FUNCTION_BLOCK "HF3_FJPG_FB2771"	// FB 2771
VERSION : 0.1
VAR
  PT : TIME  := T#45S;
  AP22_WP14 : FB 2772;
END_VAR
BEGIN
NETWORK
TITLE = AP22-wp14
      A     "EPS11_QJSS_UEF_Opd";
      =     L 0.0;
      BLD   103;
      A     "EPS11_QJSS_UEB_Opd";
      =     L 0.1;
      BLD   103;
      A     "EPS11_QJSS_DHF_Opd";
      =     L 0.2;
      BLD   103;
      A     DB7004.DBX 2630.0;
      =     L 0.4;
      BLD   103;
      A     DB7004.DBX 2630.1;
      =     L 0.5;
      BLD   103;
      BLD   14;
      =     L 7.0;
      L     DINO;
      T     LW 5;
      CDB;
      OPN   DI [LW 5];
      TAR2  LD 1;
      OPN   DI 6001;
      L     DIW 170;
      OPN   DI [LW 5];
      T     #AP22_WP14.SCtrl;
      OPN   DI 7004;
      L     DIW 840;
      OPN   DI [LW 5];
      T     #AP22_WP14.H_P_ALL_Ctrl;
      A     L 0.0;
      =     #AP22_WP14.DI_LR;
      A     L 0.1;
      =     #AP22_WP14.DI_Run;
      A     L 0.2;
      =     #AP22_WP14.DI_Stp;
      A     L 0.4;
      =     #AP22_WP14.FireAlarm;
      A     L 0.5;
      =     #AP22_WP14.BlockAlarm;
      BLD   11;
      L     W#16#1002;
      T     LW 10;
      L     2;
      T     LW 12;
      L     7004;
      T     LW 14;
      L     P#DBX 592.0;
      T     LD 16;
      L     W#16#1002;
      T     LW 20;
      L     2;
      T     LW 22;
      L     DINO;
      T     LW 24;
      +AR2  P#12.0;
      TAR2;
      LAR2  LD 1;
      T     LD 26;
      UC    "BLKMOV";
      {     P#L 10.0, P#L 8.0, P#L 20.0 };
      BLD   11;
      L     W#16#1002;
      T     LW 10;
      L     2;
      T     LW 12;
      L     7004;
      T     LW 14;
      L     P#DBX 966.0;
      T     LD 16;
      L     W#16#1002;
      T     LW 20;
      L     2;
      T     LW 22;
      L     DINO;
      T     LW 24;
      +AR2  P#14.0;
      TAR2;
      LAR2  LD 1;
      T     LD 26;
      UC    "BLKMOV";
      {     P#L 10.0, P#L 8.0, P#L 20.0 };
      L     DBD [AR2,P#0.0];
      T     #AP22_WP14.PT1;
      +AR2  P#4.0;
      UC    "HF3_FJPG_FB2772";
      LAR2  LD 1;
      A     #AP22_WP14.DO_Run;
      =     Q 2.0;
      A     #AP22_WP14.DO_Stp;
      =     Q 2.1;
      L     #AP22_WP14.ToHMI;
      OPN   DI 6002;
      T     DIW 1110;
      OPN   DI [LW 5];
      CDB;
      BLD   15;
      NOP   0;
NETWORK
TITLE = AP_B02
END_FUNCTION_BLOCK

FUNCTION_BLOCK "HF3_FJPG_FB2772"	// FB 2772
VERSION : 0.1
VAR_INPUT
  SCtrl : WORD ;	//0.单控1.模控2.单控启动3.单控停止5.超时复位11.运行次数清零12.故障清零13.
  H_P_ALL_Ctrl : WORD ;	//全局命令
  DI_LR : BOOL ;	//远程/就地
  DI_Run : BOOL ;	//风机盘管运行反馈
  DI_Stp : BOOL ;	//风机盘管停止反馈
  Stop : BOOL ;	//连锁信号
  FireAlarm : BOOL ;	//火灾信号
  BlockAlarm : BOOL ;	//阻塞信号
  MCtrl : ARRAY  [0 .. 3 ] OF //模式控制
  BOOL ;
  Mode : ARRAY  [0 .. 15 ] OF //模式执行状态
  BOOL ;
  ALL : ARRAY  [0 .. 15 ] OF //单系统命令
  BOOL ;
  PT1 : TIME ;	//设备动作超时
END_VAR
VAR_OUTPUT
  DO_Run : BOOL ;	//开阀控制
  DO_Stp : BOOL ;	//关阀控制
  ToHMI : WORD ;	//给上位信号
END_VAR
VAR
  SCtrl_Temp : ARRAY  [0 .. 15 ] OF //1.模控2.单控启动3.单控停止5.超时复位11.运行次数清零12.故障清零13.
  BOOL ;
  DI_Temp : ARRAY  [0 .. 15 ] OF BOOL ;
  DO_Temp : ARRAY  [0 .. 15 ] OF BOOL ;
  H_P_ALL_Ctrl_Temp : ARRAY  [0 .. 15 ] OF BOOL ;
  Ctrl : ARRAY  [0 .. 15 ] OF BOOL ;
  TON1 : SFB 4;
  SFlag : BOOL ;
  QTout : BOOL ;
  Timeout : BOOL ;	//设备动作超时
  Refuse : BOOL ;	//模式不符
  McFlag : BOOL ;	//检修牌
END_VAR
BEGIN
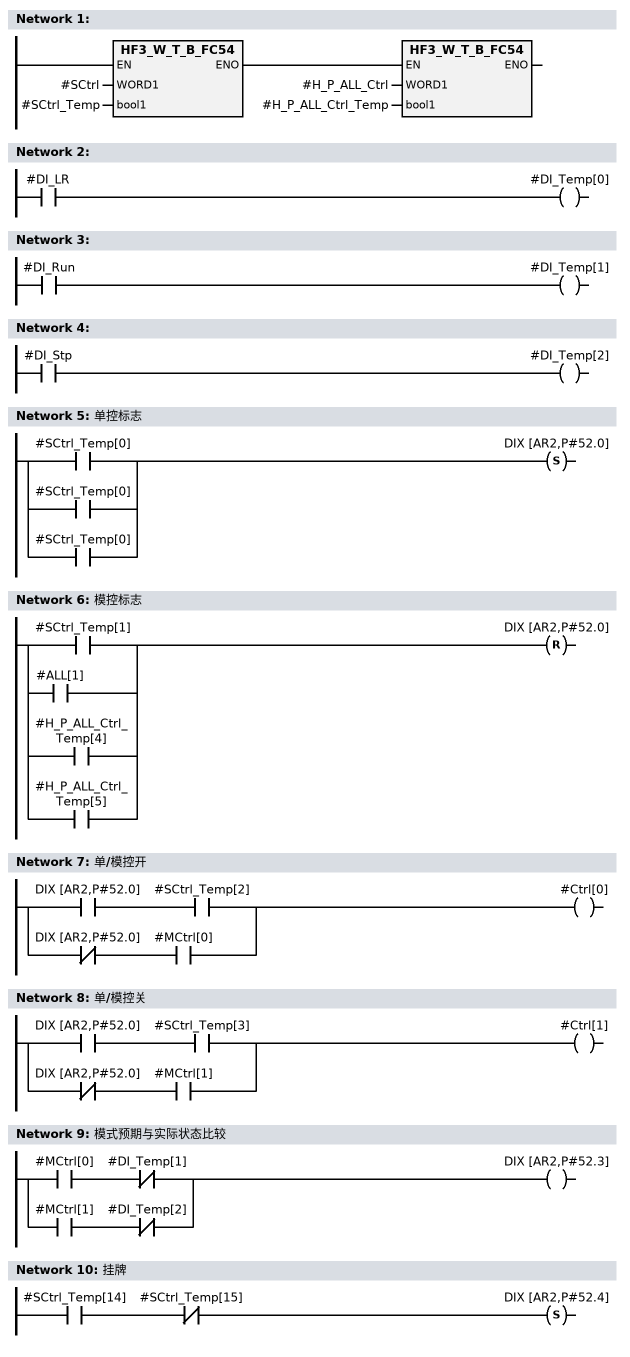
NETWORK
TITLE =
      A(;
      CALL  "HF3_W_T_B_FC54" (
           WORD1                    := #SCtrl,
           bool1                    := #SCtrl_Temp);
      A     BR;
      );
      JNB   _001;
      CALL  "HF3_W_T_B_FC54" (
           WORD1                    := #H_P_ALL_Ctrl,
           bool1                    := #H_P_ALL_Ctrl_Temp);
_001: NOP   0;
NETWORK
TITLE =
      A     #DI_LR;
      =     #DI_Temp[0];
NETWORK
TITLE =
      A     #DI_Run;
      =     #DI_Temp[1];
NETWORK
TITLE =
      A     #DI_Stp;
      =     #DI_Temp[2];
NETWORK
TITLE = 单控标志
      O     #SCtrl_Temp[0];
      O     #SCtrl_Temp[0];
      O     #SCtrl_Temp[0];
      S     DIX [AR2,P#52.0];
NETWORK
TITLE = 模控标志
      O     #SCtrl_Temp[1];
      O     #ALL[1];
      O     #H_P_ALL_Ctrl_Temp[4];
      O     #H_P_ALL_Ctrl_Temp[5];
      R     DIX [AR2,P#52.0];
NETWORK
TITLE = 单/模控开
      A     DIX [AR2,P#52.0];
      A     #SCtrl_Temp[2];
      O;
      AN    DIX [AR2,P#52.0];
      A     #MCtrl[0];
      =     #Ctrl[0];
NETWORK
TITLE = 单/模控关
      A     DIX [AR2,P#52.0];
      A     #SCtrl_Temp[3];
      O;
      AN    DIX [AR2,P#52.0];
      A     #MCtrl[1];
      =     #Ctrl[1];
NETWORK
TITLE = 模式预期与实际状态比较
      A     #MCtrl[0];
      AN    #DI_Temp[1];
      O;
      A     #MCtrl[1];
      AN    #DI_Temp[2];
      =     DIX [AR2,P#52.3];
NETWORK
TITLE = 挂牌
      A     #SCtrl_Temp[14];
      AN    #SCtrl_Temp[15];
      S     DIX [AR2,P#52.4];
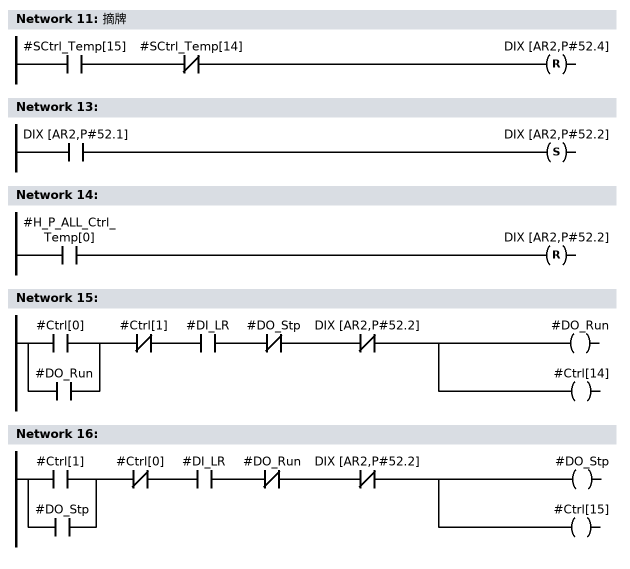
NETWORK
TITLE = 摘牌
      A     #SCtrl_Temp[15];
      AN    #SCtrl_Temp[14];
      R     DIX [AR2,P#52.4];
NETWORK
TITLE =
      A(;
      O     #Ctrl[14];
      O     #Ctrl[15];
      );
      =     L 0.0;
      BLD   103;
      BLD   16;
      =     L 7.0;
      L     DINO;
      T     LW 5;
      CDB;
      OPN   DI [LW 5];
      TAR2  LD 1;
      A     L 0.0;
      =     DIX [AR2,P#30.0];
      L     L#5000;
      T     DID [AR2,P#32.0];
      +AR2  P#30.0;
      UC    "TON";
      LAR2  LD 1;
      A     DIX [AR2,P#36.0];
      =     DBX [AR2,P#52.1];
      CDB;
      BLD   17;
      NOP   0;
NETWORK
TITLE =
      A     DIX [AR2,P#52.1];
      S     DIX [AR2,P#52.2];
NETWORK
TITLE =
      A     #H_P_ALL_Ctrl_Temp[0];
      R     DIX [AR2,P#52.2];
NETWORK
TITLE =
      A(;
      O     #Ctrl[0];
      O     #DO_Run;
      );
      AN    #Ctrl[1];
      A     #DI_LR;
      AN    #DO_Stp;
      AN    DIX [AR2,P#52.2];
      =     #DO_Run;
      =     #Ctrl[14];
NETWORK
TITLE =
      A(;
      O     #Ctrl[1];
      O     #DO_Stp;
      );
      AN    #Ctrl[0];
      A     #DI_LR;
      AN    #DO_Run;
      AN    DIX [AR2,P#52.2];
      =     #DO_Stp;
      =     #Ctrl[15];
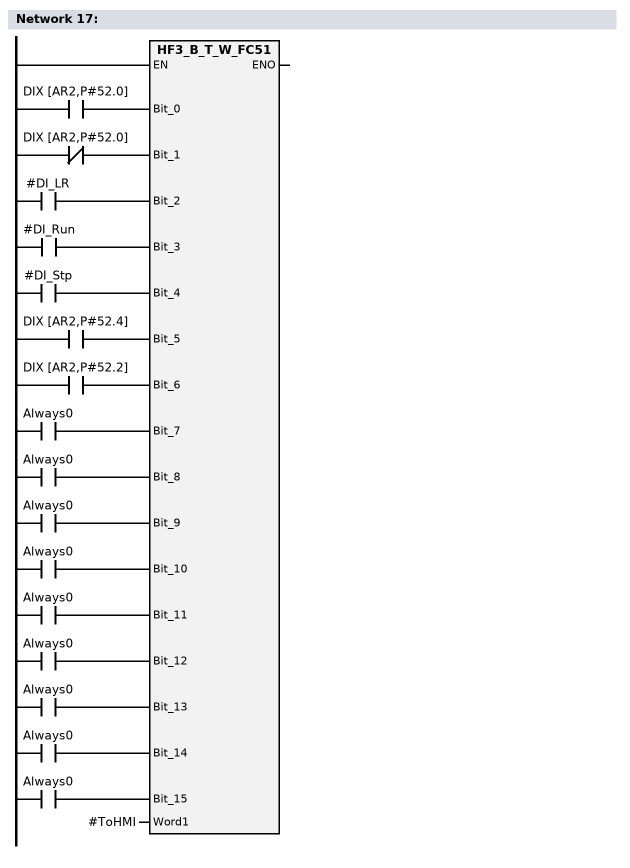
NETWORK
TITLE =
      A     DIX [AR2,P#52.0];
      =     L 0.0;
      BLD   103;
      AN    DIX [AR2,P#52.0];
      =     L 0.1;
      BLD   103;
      A     #DI_LR;
      =     L 0.2;
      BLD   103;
      A     #DI_Run;
      =     L 0.3;
      BLD   103;
      A     #DI_Stp;
      =     L 0.4;
      BLD   103;
      A     DIX [AR2,P#52.4];
      =     L 0.5;
      BLD   103;
      A     DIX [AR2,P#52.2];
      =     L 0.6;
      BLD   103;
      A     "Always0";
      =     L 0.7;
      BLD   103;
      A     "Always0";
      =     L 1.0;
      BLD   103;
      A     "Always0";
      =     L 1.1;
      BLD   103;
      A     "Always0";
      =     L 1.2;
      BLD   103;
      A     "Always0";
      =     L 1.3;
      BLD   103;
      A     "Always0";
      =     L 1.4;
      BLD   103;
      A     "Always0";
      =     L 1.5;
      BLD   103;
      A     "Always0";
      =     L 1.6;
      BLD   103;
      A     "Always0";
      =     L 1.7;
      BLD   103;
      CALL  "HF3_B_T_W_FC51" (
           Bit_0                    := L 0.0,
           Bit_1                    := L 0.1,
           Bit_2                    := L 0.2,
           Bit_3                    := L 0.3,
           Bit_4                    := L 0.4,
           Bit_5                    := L 0.5,
           Bit_6                    := L 0.6,
           Bit_7                    := L 0.7,
           Bit_8                    := L 1.0,
           Bit_9                    := L 1.1,
           Bit_10                   := L 1.2,
           Bit_11                   := L 1.3,
           Bit_12                   := L 1.4,
           Bit_13                   := L 1.5,
           Bit_14                   := L 1.6,
           Bit_15                   := L 1.7,
           Word1                    := #ToHMI);
      NOP   0;
END_FUNCTION_BLOCK

FUNCTION_BLOCK "HF3_XFDF_FB2781"	// FB 2781
VERSION : 0.1
VAR
  PT : TIME  := T#1M;
  XFDF_B1 : FB 2782;
  XFDF_B2 : FB 2782;
END_VAR
BEGIN
NETWORK
TITLE = XFDF_B1
      A     "EPS11_QJSS_DHB_opd";
      =     L 0.0;
      BLD   103;
      A     I 2.4;
      =     L 0.1;
      BLD   103;
      A     I 2.5;
      =     L 0.2;
      BLD   103;
      A     I 2.6;
      =     L 0.3;
      BLD   103;
      BLD   14;
      =     L 7.0;
      L     DINO;
      T     LW 5;
      CDB;
      OPN   DI [LW 5];
      TAR2  LD 1;
      OPN   DI 6001;
      L     DIW 172;
      OPN   DI [LW 5];
      T     #XFDF_B1.SCtrl;
      A     L 0.0;
      =     #XFDF_B1.XFDF_DI_LR;
      A     L 0.1;
      =     #XFDF_B1.XFDF_DI_Opd;
      A     L 0.2;
      =     #XFDF_B1.XFDF_DI_Cld;
      A     L 0.3;
      =     #XFDF_B1.XFDF_DI_GFlt;
      OPN   DI 7004;
      L     DIW 840;
      OPN   DI [LW 5];
      T     #XFDF_B1.H_P_All_Ctrl;
      L     DBD [AR2,P#0.0];
      T     #XFDF_B1.PT;
      +AR2  P#4.0;
      UC    "HF2_XVDF_FB2782";
      LAR2  LD 1;
      A     #XFDF_B1.XFDF_DO_Opn;
      =     Q 2.2;
      A     #XFDF_B1.XFDF_DO_Cls;
      =     Q 2.3;
      L     #XFDF_B1.ToHMI;
      OPN   DI 6002;
      T     DIW 1112;
      OPN   DI [LW 5];
      CDB;
      BLD   15;
      NOP   0;
NETWORK
TITLE = XFDF_B2
      A     "SDPH_A1_LR";
      =     L 0.0;
      BLD   103;
      A     "SDPH_K4_A1_LR";
      =     L 0.1;
      BLD   103;
      A     "YC_A_Alarm";
      =     L 0.2;
      BLD   103;
      A     "JH_A_Run";
      =     L 0.3;
      BLD   103;
      BLD   14;
      =     L 7.0;
      L     DINO;
      T     LW 5;
      CDB;
      OPN   DI [LW 5];
      TAR2  LD 1;
      OPN   DI 6001;
      L     DIW 174;
      OPN   DI [LW 5];
      T     DIW [AR2,P#80.0];
      A     L 0.0;
      =     DIX [AR2,P#82.0];
      A     L 0.1;
      =     DIX [AR2,P#82.1];
      A     L 0.2;
      =     DIX [AR2,P#82.2];
      A     L 0.3;
      =     DIX [AR2,P#82.3];
      OPN   DI 7004;
      L     DIW 840;
      OPN   DI [LW 5];
      T     DIW [AR2,P#84.0];
      L     DBD [AR2,P#0.0];
      T     DID [AR2,P#86.0];
      +AR2  P#80.0;
      UC    "HF2_XVDF_FB2782";
      LAR2  LD 1;
      A     DIX [AR2,P#90.0];
      =     "EPS11_QJSS_UEF_opn";
      A     DIX [AR2,P#90.1];
      =     "EPS11_QJSS_UEB_opn";
      L     DIW [AR2,P#92.0];
      OPN   DI 6002;
      T     DIW 1114;
      OPN   DI [LW 5];
      CDB;
      BLD   15;
      NOP   0;
END_FUNCTION_BLOCK

FUNCTION_BLOCK "HF2_XVDF_FB2782"	// FB 2782
TITLE = 手电一体蝶阀功能块
//手电一体蝶阀功能块
VERSION : 0.1
VAR_INPUT
  SCtrl : WORD ;	//ISCS控制命令
  XFDF_DI_LR : BOOL ;	//蝶阀远程就地状态
  XFDF_DI_Opd : BOOL ;	//蝶阀开状态
  XFDF_DI_Cld : BOOL ;	//蝶阀关状态
  XFDF_DI_GFlt : BOOL ;	//蝶阀综合故障状态
  H_P_All_Ctrl : WORD ;	//全局命令
  PT : TIME ;	//控制超时时间
END_VAR
VAR_OUTPUT
  XFDF_DO_Opn : BOOL ;	//开阀输出控制
  XFDF_DO_Cls : BOOL ;	//关阀输出控制
  ToHMI : WORD ;	//反馈上位信息
END_VAR
VAR
  Ton1_1 : SFB 4;
  Ton1_2 : SFB 4;
  SingTout : BOOL ;
  Timeout : BOOL ;
  DI_Temp : ARRAY  [0 .. 15 ] OF BOOL ;
  DO_Temp : ARRAY  [0 .. 15 ] OF BOOL ;
  Ctrl : ARRAY  [0 .. 15 ] OF BOOL ;
  SCtrl_Temp : ARRAY  [0 .. 15 ] OF BOOL ;
  Latch : ARRAY  [0 .. 7 ] OF BOOL ;
  QTout : BOOL ;
  H_P_All_Ctrl_Temp : ARRAY  [0 .. 15 ] OF BOOL ;
  McFlag : BOOL ;
END_VAR
BEGIN
NETWORK
TITLE =
      A(;
      BLD   1;
      =     L 4.0;
      TAR2  LD 0;
      L     #SCtrl;
      T     LW 5;
      L     DINO;
      T     LW 7;
      +AR2  P#66.0;
      TAR2;
      LAR2  LD 0;
      T     LD 9;
      UC    "HF3_W_T_B_FC54";
      {     P#L 5.0, P#L 7.0 };
      LAR2  LD 0;
      BLD   2;
      A     BR;
      );
      JNB   _001;
      BLD   1;
      =     L 4.0;
      TAR2  LD 0;
      L     #H_P_All_Ctrl;
      T     LW 5;
      L     DINO;
      T     LW 7;
      +AR2  P#72.0;
      TAR2;
      LAR2  LD 0;
      T     LD 9;
      UC    "HF3_W_T_B_FC54";
      {     P#L 5.0, P#L 7.0 };
      LAR2  LD 0;
      BLD   2;
_001: NOP   0;
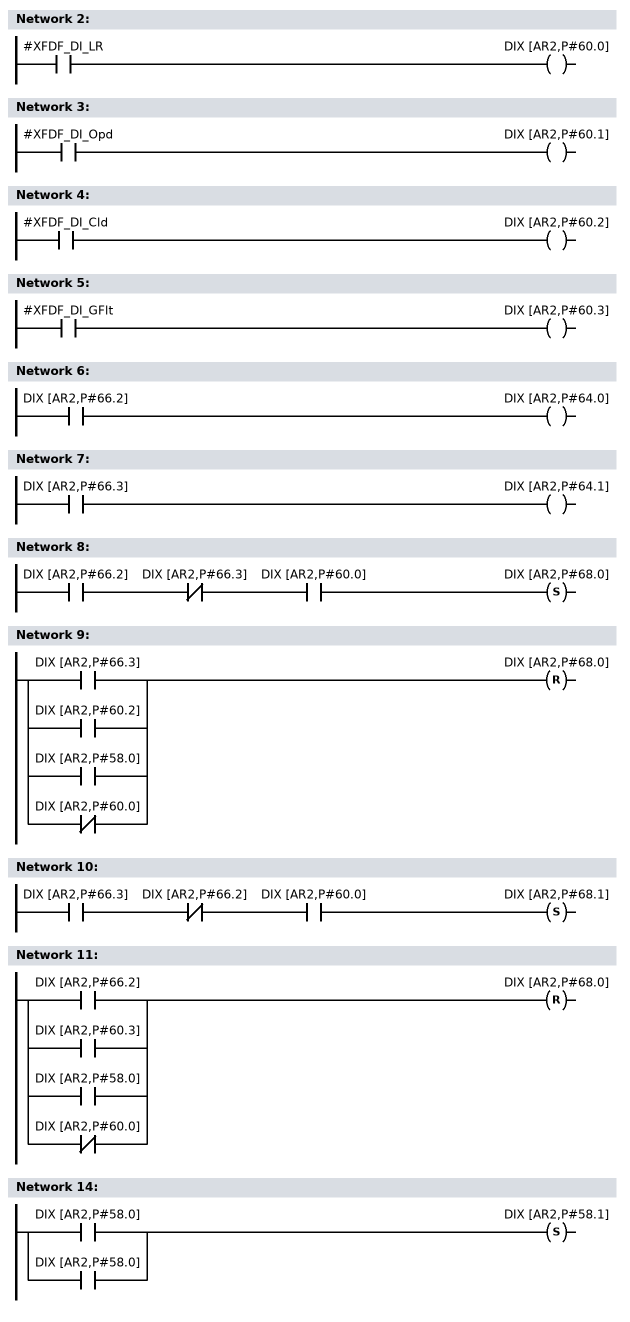
NETWORK
TITLE =
      A     #XFDF_DI_LR;
      =     DIX [AR2,P#60.0];
NETWORK
TITLE =
      A     #XFDF_DI_Opd;
      =     DIX [AR2,P#60.1];
NETWORK
TITLE =
      A     #XFDF_DI_Cld;
      =     DIX [AR2,P#60.2];
NETWORK
TITLE =
      A     #XFDF_DI_GFlt;
      =     DIX [AR2,P#60.3];
NETWORK
TITLE =
      A     DIX [AR2,P#66.2];
      =     DIX [AR2,P#64.0];
NETWORK
TITLE =
      A     DIX [AR2,P#66.3];
      =     DIX [AR2,P#64.1];
NETWORK
TITLE =
      A     DIX [AR2,P#66.2];
      AN    DIX [AR2,P#66.3];
      A     DIX [AR2,P#60.0];
      S     DIX [AR2,P#68.0];
NETWORK
TITLE =
      O     DIX [AR2,P#66.3];
      O     DIX [AR2,P#60.2];
      O     DIX [AR2,P#58.0];
      ON    DIX [AR2,P#60.0];
      R     DIX [AR2,P#68.0];
NETWORK
TITLE =
      A     DIX [AR2,P#66.3];
      AN    DIX [AR2,P#66.2];
      A     DIX [AR2,P#60.0];
      S     DIX [AR2,P#68.1];
NETWORK
TITLE =
      O     DIX [AR2,P#66.2];
      O     DIX [AR2,P#60.3];
      O     DIX [AR2,P#58.0];
      ON    DIX [AR2,P#60.0];
      R     DIX [AR2,P#68.0];
NETWORK
TITLE =
      A(;
      A     DIX [AR2,P#68.0];
      AN    DIX [AR2,P#60.1];
      O;
      A     DIX [AR2,P#68.1];
      AN    DIX [AR2,P#60.2];
      );
      =     L 0.0;
      BLD   103;
      BLD   16;
      =     L 7.0;
      L     DINO;
      T     LW 5;
      CDB;
      OPN   DI [LW 5];
      TAR2  LD 1;
      A     L 0.0;
      =     DIX [AR2,P#14.0];
      L     DBD [AR2,P#6.0];
      T     DID [AR2,P#16.0];
      +AR2  P#14.0;
      UC    "TON";
      LAR2  LD 1;
      A     DIX [AR2,P#20.0];
      =     DBX [AR2,P#58.0];
      CDB;
      BLD   17;
      NOP   0;
NETWORK
TITLE =
      A(;
      O     DIX [AR2,P#62.0];
      O     DIX [AR2,P#62.1];
      );
      =     L 0.0;
      BLD   103;
      BLD   16;
      =     L 7.0;
      L     DINO;
      T     LW 5;
      CDB;
      OPN   DI [LW 5];
      TAR2  LD 1;
      A     L 0.0;
      =     DIX [AR2,P#14.0];
      L     DBD [AR2,P#6.0];
      T     DID [AR2,P#16.0];
      +AR2  P#14.0;
      UC    "TON";
      LAR2  LD 1;
      A     DIX [AR2,P#20.0];
      =     DBX [AR2,P#70.0];
      CDB;
      BLD   17;
      NOP   0;
NETWORK
TITLE =
      O     DIX [AR2,P#58.0];
      O     DIX [AR2,P#58.0];
      S     DIX [AR2,P#58.1];
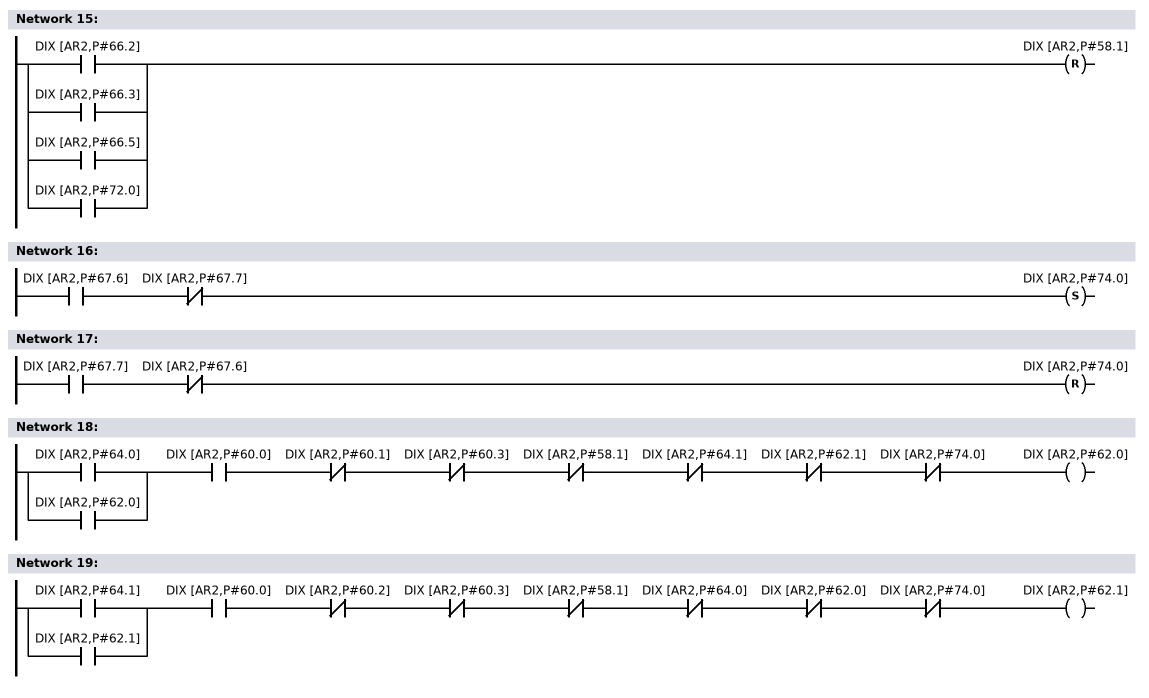
NETWORK
TITLE =
      O     DIX [AR2,P#66.2];
      O     DIX [AR2,P#66.3];
      O     DIX [AR2,P#66.5];
      O     DIX [AR2,P#72.0];
      R     DIX [AR2,P#58.1];
NETWORK
TITLE =
      A     DIX [AR2,P#67.6];
      AN    DIX [AR2,P#67.7];
      S     DIX [AR2,P#74.0];
NETWORK
TITLE =
      A     DIX [AR2,P#67.7];
      AN    DIX [AR2,P#67.6];
      R     DIX [AR2,P#74.0];
NETWORK
TITLE =
      A(;
      O     DIX [AR2,P#64.0];
      O     DIX [AR2,P#62.0];
      );
      A     DIX [AR2,P#60.0];
      AN    DIX [AR2,P#60.1];
      AN    DIX [AR2,P#60.3];
      AN    DIX [AR2,P#58.1];
      AN    DIX [AR2,P#64.1];
      AN    DIX [AR2,P#62.1];
      AN    DIX [AR2,P#74.0];
      =     DIX [AR2,P#62.0];
NETWORK
TITLE =
      A(;
      O     DIX [AR2,P#64.1];
      O     DIX [AR2,P#62.1];
      );
      A     DIX [AR2,P#60.0];
      AN    DIX [AR2,P#60.2];
      AN    DIX [AR2,P#60.3];
      AN    DIX [AR2,P#58.1];
      AN    DIX [AR2,P#64.0];
      AN    DIX [AR2,P#62.0];
      AN    DIX [AR2,P#74.0];
      =     DIX [AR2,P#62.1];
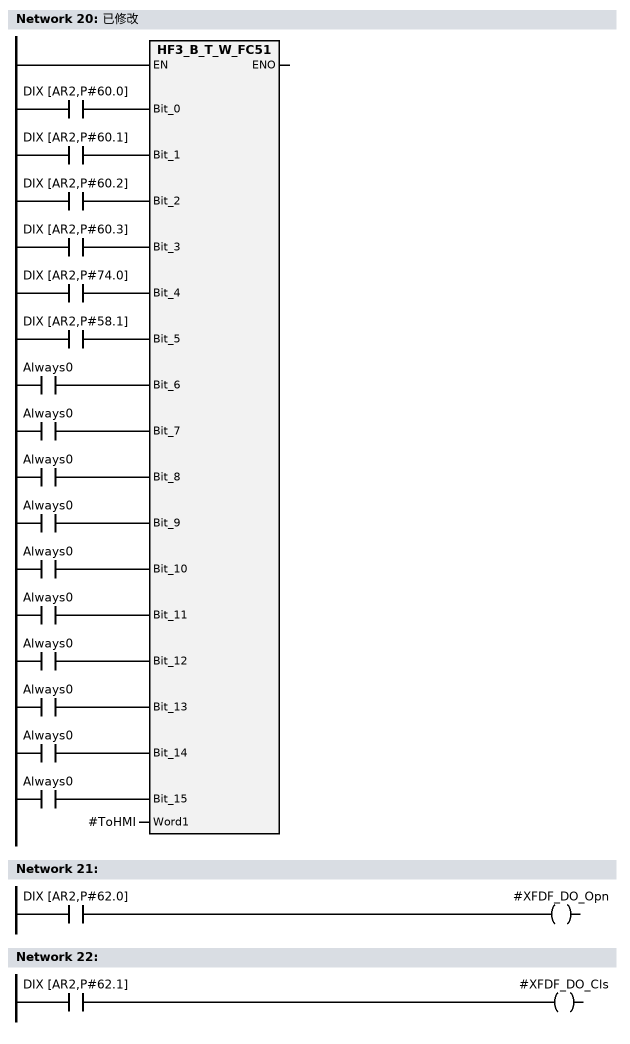
NETWORK
TITLE = 已修改
      A     DIX [AR2,P#60.0];
      =     L 0.0;
      BLD   103;
      A     DIX [AR2,P#60.1];
      =     L 0.1;
      BLD   103;
      A     DIX [AR2,P#60.2];
      =     L 0.2;
      BLD   103;
      A     DIX [AR2,P#60.3];
      =     L 0.3;
      BLD   103;
      A     DIX [AR2,P#74.0];
      =     L 0.4;
      BLD   103;
      A     DIX [AR2,P#58.1];
      =     L 0.5;
      BLD   103;
      A     "Always0";
      =     L 0.6;
      BLD   103;
      A     "Always0";
      =     L 0.7;
      BLD   103;
      A     "Always0";
      =     L 1.0;
      BLD   103;
      A     "Always0";
      =     L 1.1;
      BLD   103;
      A     "Always0";
      =     L 1.2;
      BLD   103;
      A     "Always0";
      =     L 1.3;
      BLD   103;
      A     "Always0";
      =     L 1.4;
      BLD   103;
      A     "Always0";
      =     L 1.5;
      BLD   103;
      A     "Always0";
      =     L 1.6;
      BLD   103;
      A     "Always0";
      =     L 1.7;
      BLD   103;
      CALL  "HF3_B_T_W_FC51" (
           Bit_0                    := L 0.0,
           Bit_1                    := L 0.1,
           Bit_2                    := L 0.2,
           Bit_3                    := L 0.3,
           Bit_4                    := L 0.4,
           Bit_5                    := L 0.5,
           Bit_6                    := L 0.6,
           Bit_7                    := L 0.7,
           Bit_8                    := L 1.0,
           Bit_9                    := L 1.1,
           Bit_10                   := L 1.2,
           Bit_11                   := L 1.3,
           Bit_12                   := L 1.4,
           Bit_13                   := L 1.5,
           Bit_14                   := L 1.6,
           Bit_15                   := L 1.7,
           Word1                    := #ToHMI);
      NOP   0;
NETWORK
TITLE =
      A     DIX [AR2,P#62.0];
      =     #XFDF_DO_Opn;
NETWORK
TITLE =
      A     DIX [AR2,P#62.1];
      =     #XFDF_DO_Cls;
END_FUNCTION_BLOCK

FUNCTION_BLOCK "HF3_EPS_WLE_FB2791"	// FB 2791
TITLE = 区间疏散指示系统   一个控制系统含4条控制回路
//
//EPSA_DEF_OpnQ       6.2BOOL下行尾前向控
//EPSA_DEF_OpdI      24.2BOOL下行尾前向馈
//EPSA_DEB_OpnQ       6.3BOOL下行尾后向控
//EPSA_DEB_opdI      24.3BOOL下行尾后向馈
//
VERSION : 0.1
VAR
  WLEB_1 : FB 2792;
  WLEB_2 : FB 2792;
  WLEB_3 : FB 2792;
  WLEB_4 : FB 2792;
  PT_WLE : TIME  := T#45S;
END_VAR
BEGIN
NETWORK
TITLE = 回路一
      A     "EPS11_QJSS_UEF_Opd";
      =     L 0.0;
      BLD   103;
      BLD   14;
      =     L 7.0;
      L     DINO;
      T     LW 5;
      CDB;
      OPN   DI [LW 5];
      TAR2  LD 1;
      OPN   DI 6003;
      L     DIW 102;
      OPN   DI [LW 5];
      T     #WLEB_1.SCtrl;
      A     L 0.0;
      =     #WLEB_1.iOn;
      L     DBD [AR2,P#336.0];
      T     #WLEB_1.PT;
      OPN   DI 7005;
      L     DIW 312;
      OPN   DI [LW 5];
      T     #WLEB_1.H_P_All_Ctrl;
      +AR2  P#0.0;
      UC    "HF3_EPS_WLE_FB2792";
      LAR2  LD 1;
      A     #WLEB_1.qOn;
      =     "EPS11_QJSS_UEF_opn";
      L     #WLEB_1.ToHMI;
      OPN   DI 6004;
      T     DIW 772;
      OPN   DI [LW 5];
      CDB;
      BLD   15;
      NOP   0;
NETWORK
TITLE = 回路二
      A     "EPS11_QJSS_UEB_Opd";
      =     L 0.0;
      BLD   103;
      A     "Always0";
      =     L 0.1;
      BLD   103;
      BLD   14;
      =     L 7.0;
      L     DINO;
      T     LW 5;
      CDB;
      OPN   DI [LW 5];
      TAR2  LD 1;
      OPN   DI 6003;
      L     DIW 104;
      OPN   DI [LW 5];
      T     DIW [AR2,P#84.0];
      A     L 0.0;
      =     DIX [AR2,P#86.0];
      L     DBD [AR2,P#336.0];
      T     DID [AR2,P#92.0];
      A     L 0.1;
      =     DIX [AR2,P#98.0];
      OPN   DI 7005;
      L     DIW 312;
      OPN   DI [LW 5];
      T     DIW [AR2,P#100.0];
      +AR2  P#84.0;
      UC    "HF3_EPS_WLE_FB2792";
      LAR2  LD 1;
      A     DIX [AR2,P#102.0];
      =     "EPS11_QJSS_UEB_opn";
      L     DIW [AR2,P#104.0];
      OPN   DI 6004;
      T     DIW 774;
      OPN   DI [LW 5];
      CDB;
      BLD   15;
      NOP   0;
NETWORK
TITLE = 回路三
      A     "EPS11_QJSS_DHF_Opd";
      =     L 0.0;
      BLD   103;
      A     "Always0";
      =     L 0.1;
      BLD   103;
      BLD   14;
      =     L 7.0;
      L     DINO;
      T     LW 5;
      CDB;
      OPN   DI [LW 5];
      TAR2  LD 1;
      OPN   DI 6003;
      L     DIW 106;
      OPN   DI [LW 5];
      T     DIW [AR2,P#168.0];
      A     L 0.0;
      =     DIX [AR2,P#170.0];
      L     DBD [AR2,P#336.0];
      T     DID [AR2,P#176.0];
      A     L 0.1;
      =     DIX [AR2,P#182.0];
      OPN   DI 7005;
      L     DIW 312;
      OPN   DI [LW 5];
      T     DIW [AR2,P#184.0];
      +AR2  P#168.0;
      UC    "HF3_EPS_WLE_FB2792";
      LAR2  LD 1;
      A     DIX [AR2,P#186.0];
      =     "EPS11_QJSS_DHF_opn";
      L     DIW [AR2,P#188.0];
      OPN   DI 6004;
      T     DIW 776;
      OPN   DI [LW 5];
      CDB;
      BLD   15;
      NOP   0;
NETWORK
TITLE = 回路四
      A     "EPS11_QJSS_DHB_opd";
      =     L 0.0;
      BLD   103;
      A     "Always0";
      =     L 0.1;
      BLD   103;
      BLD   14;
      =     L 7.0;
      L     DINO;
      T     LW 5;
      CDB;
      OPN   DI [LW 5];
      TAR2  LD 1;
      OPN   DI 6003;
      L     DIW 108;
      OPN   DI [LW 5];
      T     DIW [AR2,P#252.0];
      A     L 0.0;
      =     DIX [AR2,P#254.0];
      L     DBD [AR2,P#336.0];
      T     DID [AR2,P#260.0];
      A     L 0.1;
      =     DIX [AR2,P#266.0];
      OPN   DI 7005;
      L     DIW 312;
      OPN   DI [LW 5];
      T     DIW [AR2,P#268.0];
      +AR2  P#252.0;
      UC    "HF3_EPS_WLE_FB2792";
      LAR2  LD 1;
      A     DIX [AR2,P#270.0];
      =     "EPS11_QJSS_DHB_opn";
      L     DIW [AR2,P#272.0];
      OPN   DI 6004;
      T     DIW 778;
      OPN   DI [LW 5];
      CDB;
      BLD   15;
      NOP   0;
END_FUNCTION_BLOCK

FUNCTION_BLOCK "HF3_EPS_WLE_FB2792"	// FB 2792
VERSION : 0.1
VAR_INPUT
  SCtrl : WORD ;	//点动控制
  iOn : BOOL ;	//开反馈
  MCtrl : ARRAY  [0 .. 3 ] OF //模式控制
  BOOL ;
  Mode : ARRAY  [0 .. 15 ] OF //模式执行状态
  BOOL ;
  PT : TIME ;	//设备动作超时时间
  ALL : ARRAY  [0 .. 15 ] OF //单系统命令
  BOOL ;
  Fire_RE : BOOL ;	//火灾上升沿
  H_P_All_Ctrl : WORD ;	//全局命令
END_VAR
VAR_OUTPUT
  qOn : BOOL ;	//开控制命令
  ToHMI : WORD ;	//给上位状态信息
END_VAR
VAR
  Ctrl : ARRAY  [0 .. 15 ] OF BOOL ;
  Latch : ARRAY  [0 .. 15 ] OF BOOL ;
  SFlag : BOOL ;	//单控标志
  SingTout : BOOL ;	//单控超时
  Timeout : BOOL ;	//设备动作超时
  Refuse : BOOL ;	//模式不符
  RT1 : REAL ;	//累计运行时间（天)
  Maintenance : BOOL ;	//挂牌检修
  TON1 : SFB 4;
  Sctrl_temp : ARRAY  [0 .. 15 ] OF //[0]单控[1]模控[2]单控全开[3]单控小开[4]单控关阀[5]超时复位[11]运行次数清零[12]
  BOOL ;
  H_P_All_Ctrl_temp : ARRAY  [0 .. 15 ] OF BOOL ;
  ton2 : SFB 4;
  Qout : BOOL ;	//输出超时
END_VAR
VAR_TEMP
  ToHMI_temp : ARRAY  [0 .. 15 ] OF //临时状态变量
  BOOL ;
END_VAR
BEGIN
NETWORK
TITLE =
      A(;
      BLD   1;
      =     L 6.0;
      TAR2  LD 2;
      L     #SCtrl;
      T     LW 7;
      L     DINO;
      T     LW 9;
      +AR2  P#56.0;
      TAR2;
      LAR2  LD 2;
      T     LD 11;
      UC    "HF3_W_T_B_FC54";
      {     P#L 7.0, P#L 9.0 };
      LAR2  LD 2;
      BLD   2;
      A     BR;
      );
      JNB   _001;
      BLD   1;
      =     L 6.0;
      TAR2  LD 2;
      L     #H_P_All_Ctrl;
      T     LW 7;
      L     DINO;
      T     LW 9;
      +AR2  P#58.0;
      TAR2;
      LAR2  LD 2;
      T     LD 11;
      UC    "HF3_W_T_B_FC54";
      {     P#L 7.0, P#L 9.0 };
      LAR2  LD 2;
      BLD   2;
_001: NOP   0;
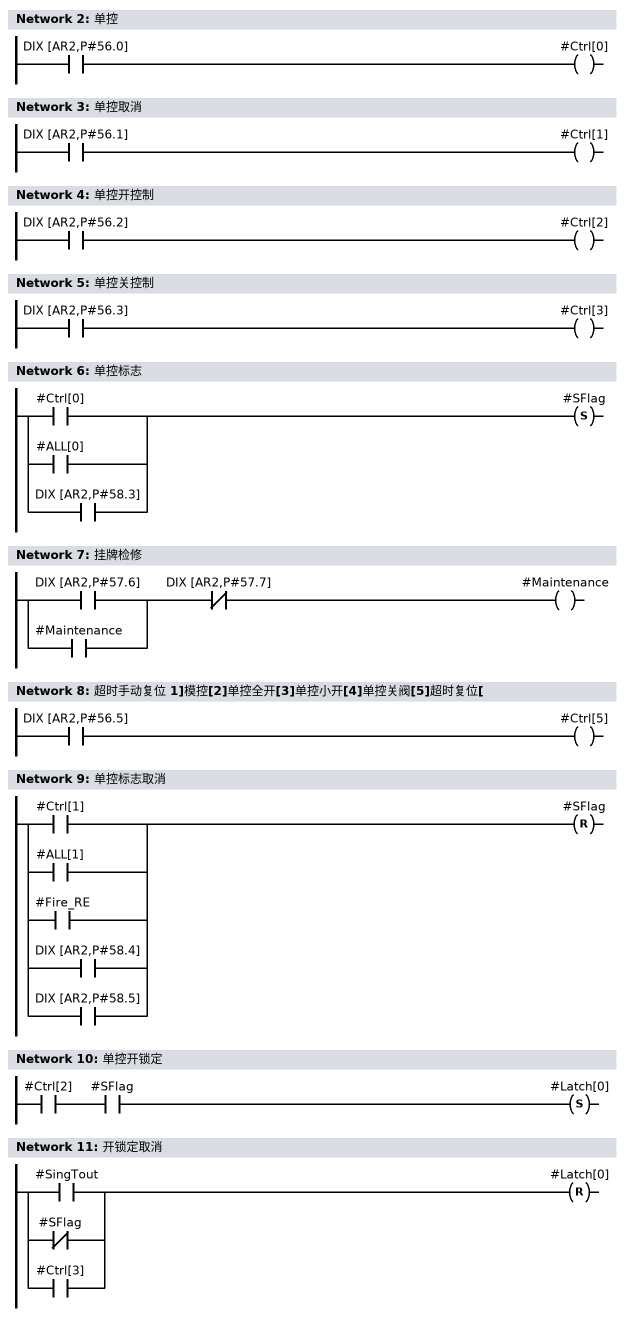
NETWORK
TITLE = 单控
      A     DIX [AR2,P#56.0];
      =     #Ctrl[0];
NETWORK
TITLE = 单控取消
      A     DIX [AR2,P#56.1];
      =     #Ctrl[1];
NETWORK
TITLE = 单控开控制
      A     DIX [AR2,P#56.2];
      =     #Ctrl[2];
NETWORK
TITLE = 单控关控制
      A     DIX [AR2,P#56.3];
      =     #Ctrl[3];
NETWORK
TITLE = 单控标志
      O     #Ctrl[0];
      O     #ALL[0];
      O     DIX [AR2,P#58.3];
      S     #SFlag;
NETWORK
TITLE = 挂牌检修
      A(;
      O     DIX [AR2,P#57.6];
      O     #Maintenance;
      );
      AN    DIX [AR2,P#57.7];
      =     #Maintenance;
NETWORK
TITLE = 超时手动复位 1]模控[2]单控全开[3]单控小开[4]单控关阀[5]超时复位[
      A     DIX [AR2,P#56.5];
      =     #Ctrl[5];
NETWORK
TITLE = 单控标志取消
      O     #Ctrl[1];
      O     #ALL[1];
      O     #Fire_RE;
      O     DIX [AR2,P#58.4];
      O     DIX [AR2,P#58.5];
      R     #SFlag;
NETWORK
TITLE = 单控开锁定
      A     #Ctrl[2];
      A     #SFlag;
      S     #Latch[0];
NETWORK
TITLE = 开锁定取消
      O     #SingTout;
      ON    #SFlag;
      O     #Ctrl[3];
      R     #Latch[0];
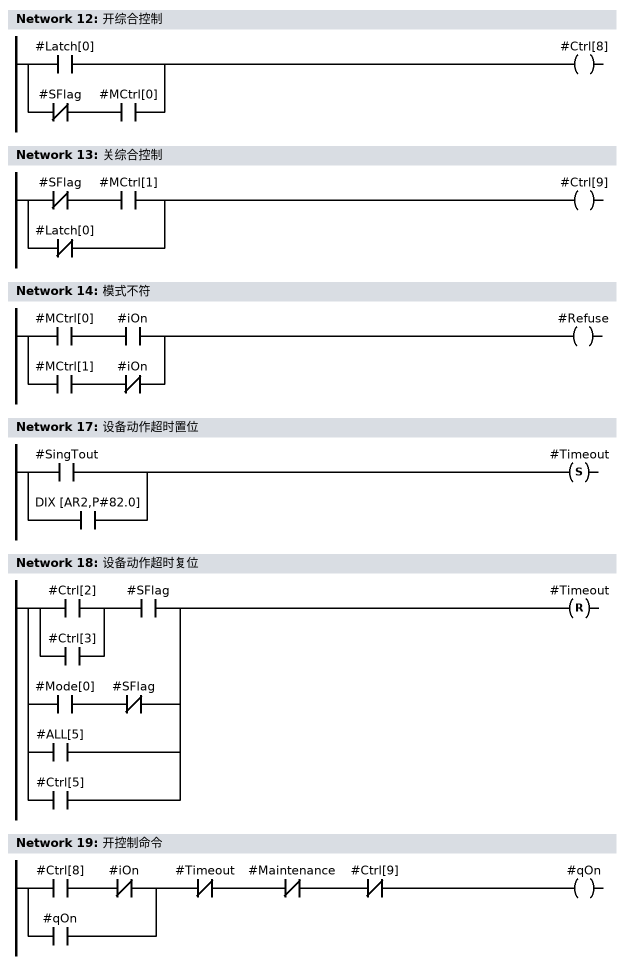
NETWORK
TITLE = 开综合控制
      O     #Latch[0];
      O;
      AN    #SFlag;
      A     #MCtrl[0];
      =     #Ctrl[8];
NETWORK
TITLE = 关综合控制
      AN    #SFlag;
      A     #MCtrl[1];
      ON    #Latch[0];
      =     #Ctrl[9];
NETWORK
TITLE = 模式不符
      A     #MCtrl[0];
      A     #iOn;
      O;
      A     #MCtrl[1];
      AN    #iOn;
      =     #Refuse;
NETWORK
TITLE = 单控超时判断
      A     #Latch[0];
      AN    #iOn;
      AN    DIX [AR2,P#56.0];
      AN    DIX [AR2,P#56.1];
      =     L 2.0;
      BLD   103;
      BLD   16;
      =     L 9.0;
      L     DINO;
      T     LW 7;
      CDB;
      OPN   DI [LW 7];
      TAR2  LD 3;
      A     L 2.0;
      =     DIX [AR2,P#34.0];
      L     DBD [AR2,P#8.0];
      T     DID [AR2,P#36.0];
      +AR2  P#34.0;
      UC    "TON";
      LAR2  LD 3;
      A     DIX [AR2,P#40.0];
      =     DBX [AR2,P#26.1];
      CDB;
      BLD   17;
      NOP   0;
NETWORK
TITLE =
      A     DIX [AR2,P#82.0];
      =     L 2.0;
      BLD   103;
      BLD   16;
      =     L 9.0;
      L     DINO;
      T     LW 7;
      CDB;
      OPN   DI [LW 7];
      TAR2  LD 3;
      A     L 2.0;
      =     DIX [AR2,P#60.0];
      L     DBD [AR2,P#8.0];
      T     DID [AR2,P#62.0];
      +AR2  P#60.0;
      UC    "TON";
      LAR2  LD 3;
      A     DIX [AR2,P#66.0];
      =     DBX [AR2,P#82.0];
      CDB;
      BLD   17;
      NOP   0;
NETWORK
TITLE = 设备动作超时置位
      O     #SingTout;
      O     DIX [AR2,P#82.0];
      S     #Timeout;
NETWORK
TITLE = 设备动作超时复位
      A(;
      O     #Ctrl[2];
      O     #Ctrl[3];
      );
      A     #SFlag;
      O;
      A     #Mode[0];
      AN    #SFlag;
      O     #ALL[5];
      O     #Ctrl[5];
      R     #Timeout;
NETWORK
TITLE = 开控制命令
      A(;
      A     #Ctrl[8];
      AN    #iOn;
      O     #qOn;
      );
      AN    #Timeout;
      AN    #Maintenance;
      AN    #Ctrl[9];
      =     #qOn;
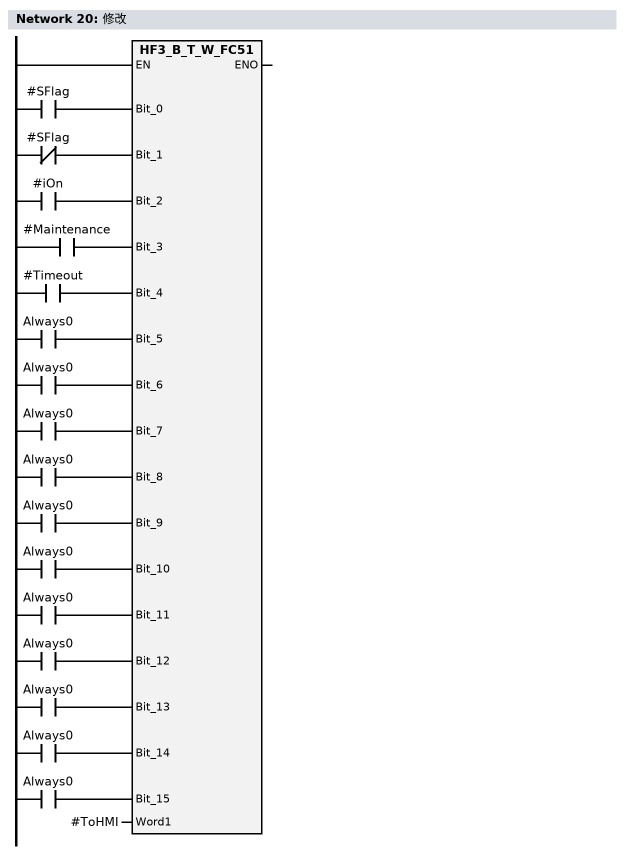
NETWORK
TITLE = 修改
      A     #SFlag;
      =     L 2.0;
      BLD   103;
      AN    #SFlag;
      =     L 2.1;
      BLD   103;
      A     #iOn;
      =     L 2.2;
      BLD   103;
      A     #Maintenance;
      =     L 2.3;
      BLD   103;
      A     #Timeout;
      =     L 2.4;
      BLD   103;
      A     "Always0";
      =     L 2.5;
      BLD   103;
      A     "Always0";
      =     L 2.6;
      BLD   103;
      A     "Always0";
      =     L 2.7;
      BLD   103;
      A     "Always0";
      =     L 3.0;
      BLD   103;
      A     "Always0";
      =     L 3.1;
      BLD   103;
      A     "Always0";
      =     L 3.2;
      BLD   103;
      A     "Always0";
      =     L 3.3;
      BLD   103;
      A     "Always0";
      =     L 3.4;
      BLD   103;
      A     "Always0";
      =     L 3.5;
      BLD   103;
      A     "Always0";
      =     L 3.6;
      BLD   103;
      A     "Always0";
      =     L 3.7;
      BLD   103;
      CALL  "HF3_B_T_W_FC51" (
           Bit_0                    := L 2.0,
           Bit_1                    := L 2.1,
           Bit_2                    := L 2.2,
           Bit_3                    := L 2.3,
           Bit_4                    := L 2.4,
           Bit_5                    := L 2.5,
           Bit_6                    := L 2.6,
           Bit_7                    := L 2.7,
           Bit_8                    := L 3.0,
           Bit_9                    := L 3.1,
           Bit_10                   := L 3.2,
           Bit_11                   := L 3.3,
           Bit_12                   := L 3.4,
           Bit_13                   := L 3.5,
           Bit_14                   := L 3.6,
           Bit_15                   := L 3.7,
           Word1                    := #ToHMI);
      NOP   0;
END_FUNCTION_BLOCK

FUNCTION_BLOCK "HF3_D_FB2801"	// FB 2801
VERSION : 0.1
VAR
  D1 : FB 2802;
  D2 : FB 2802;
END_VAR
BEGIN
NETWORK
TITLE = D1
      A     M 1.1;
      =     L 0.0;
      BLD   103;
      A     M 1.2;
      =     L 0.1;
      BLD   103;
      A     M 1.3;
      =     L 0.2;
      BLD   103;
      A     M 1.4;
      =     L 0.3;
      BLD   103;
      A     M 1.5;
      =     L 0.4;
      BLD   103;
      A     M 1.6;
      =     L 0.5;
      BLD   103;
      A     M 1.7;
      =     L 0.6;
      BLD   103;
      BLD   14;
      =     L 7.0;
      L     DINO;
      T     LW 5;
      CDB;
      OPN   DI [LW 5];
      TAR2  LD 1;
      L     MW 4;
      T     #D1.SCtrl;
      L     MW 6;
      T     #D1.H_P_ALL_Ctrl;
      A     L 0.0;
      =     #D1.DI_LR;
      A     L 0.1;
      =     #D1.DI_Opd;
      A     L 0.2;
      =     #D1.DI_Cld;
      A     L 0.3;
      =     #D1.DI_Flt;
      A     L 0.4;
      =     #D1.Stop;
      A     L 0.5;
      =     #D1.FireAlarm;
      A     L 0.6;
      =     #D1.BlockAlarm;
      +AR2  P#0.0;
      UC    "HF3_D_FB2802";
      LAR2  LD 1;
      A     #D1.DO_Opn;
      =     M 2.0;
      A     #D1.DO_Cls;
      =     M 2.1;
      L     #D1.ToHMI;
      T     MW 10;
      CDB;
      BLD   15;
      NOP   0;
NETWORK
TITLE = D2
      A     "Always0";
      =     L 0.0;
      BLD   103;
      BLD   14;
      =     L 7.0;
      L     DINO;
      T     LW 5;
      CDB;
      OPN   DI [LW 5];
      TAR2  LD 1;
      A     L 0.0;
      =     DIX [AR2,P#132.0];
      +AR2  P#128.0;
      UC    "HF3_D_FB2802";
      LAR2  LD 1;
      CDB;
      BLD   15;
      NOP   0;
END_FUNCTION_BLOCK

FUNCTION_BLOCK "HF3_D_FB2802"	// FB 2802
//[0]单控[1]模控[2]单控开阀[3]单控关阀[5]超时复位[11]运行次数清零[12]故障清零[13]
VERSION : 0.1
VAR_INPUT
  SCtrl : WORD ;
  H_P_ALL_Ctrl : WORD ;	//全局命令
  DI_LR : BOOL ;	//远程/就地
  DI_Opd : BOOL ;	//开反馈
  DI_Cld : BOOL ;	//关反馈
  DI_Flt : BOOL ;	//故障反馈
  Stop : BOOL ;	//连锁信号
  FireAlarm : BOOL ;	//火灾信号
  BlockAlarm : BOOL ;	//阻塞信号
  MCtrl : ARRAY  [0 .. 3 ] OF //模式控制
  BOOL ;
  Mode : ARRAY  [0 .. 15 ] OF //模式执行状态
  BOOL ;
  ALL : ARRAY  [0 .. 15 ] OF //单系统命令
  BOOL ;
  PT1 : TIMER ;	//设备动作超时
END_VAR
VAR_OUTPUT
  DO_Opn : BOOL ;	//开阀控制
  DO_Cls : BOOL ;	//关阀控制
  ToHMI : WORD ;	//给上位信号
  RT : INT ;	//运行时间
  SumFlt : INT ;	//故障次数
  SumRun : INT ;	//启动次数
END_VAR
VAR
  SCtrl_Temp : ARRAY  [0 .. 15 ] OF BOOL ;
  DI_Temp : ARRAY  [0 .. 15 ] OF BOOL ;
  DO_Temp : ARRAY  [0 .. 15 ] OF BOOL ;
  H_P_ALL_Ctrl_Temp : ARRAY  [0 .. 15 ] OF BOOL ;
  Ctrl : ARRAY  [0 .. 15 ] OF BOOL ;
  TON1 : SFB 4;
  TON2 : SFB 4;
  TON3 : SFB 4;
  TON4 : SFB 4;
  SFlag : BOOL ;
  QTout : BOOL ;
  Timeout : BOOL ;	//设备动作超时
  Refuse : BOOL ;	//模式不符
  McFlag : BOOL ;	//检修牌
  Latch : ARRAY  [0 .. 15 ] OF BOOL ;
  SIngTout : BOOL ;
END_VAR
BEGIN
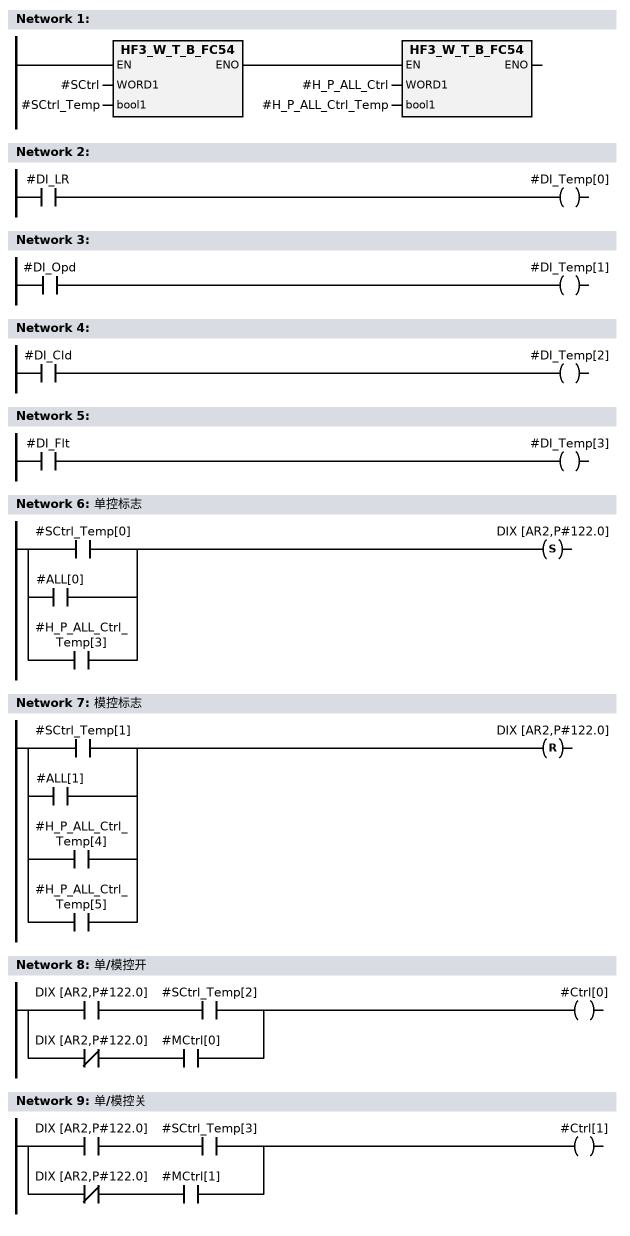
NETWORK
TITLE =
      A(;
      CALL  "HF3_W_T_B_FC54" (
           WORD1                    := #SCtrl,
           bool1                    := #SCtrl_Temp);
      A     BR;
      );
      JNB   _001;
      CALL  "HF3_W_T_B_FC54" (
           WORD1                    := #H_P_ALL_Ctrl,
           bool1                    := #H_P_ALL_Ctrl_Temp);
_001: NOP   0;
NETWORK
TITLE =
      A     #DI_LR;
      =     #DI_Temp[0];
NETWORK
TITLE =
      A     #DI_Opd;
      =     #DI_Temp[1];
NETWORK
TITLE =
      A     #DI_Cld;
      =     #DI_Temp[2];
NETWORK
TITLE =
      A     #DI_Flt;
      =     #DI_Temp[3];
NETWORK
TITLE = 单控标志
      O     #SCtrl_Temp[0];
      O     #ALL[0];
      O     #H_P_ALL_Ctrl_Temp[3];
      S     DIX [AR2,P#122.0];
NETWORK
TITLE = 模控标志
      O     #SCtrl_Temp[1];
      O     #ALL[1];
      O     #H_P_ALL_Ctrl_Temp[4];
      O     #H_P_ALL_Ctrl_Temp[5];
      R     DIX [AR2,P#122.0];
NETWORK
TITLE = 单/模控开
      A     DIX [AR2,P#122.0];
      A     #SCtrl_Temp[2];
      O;
      AN    DIX [AR2,P#122.0];
      A     #MCtrl[0];
      =     #Ctrl[0];
NETWORK
TITLE = 单/模控关
      A     DIX [AR2,P#122.0];
      A     #SCtrl_Temp[3];
      O;
      AN    DIX [AR2,P#122.0];
      A     #MCtrl[1];
      =     #Ctrl[1];
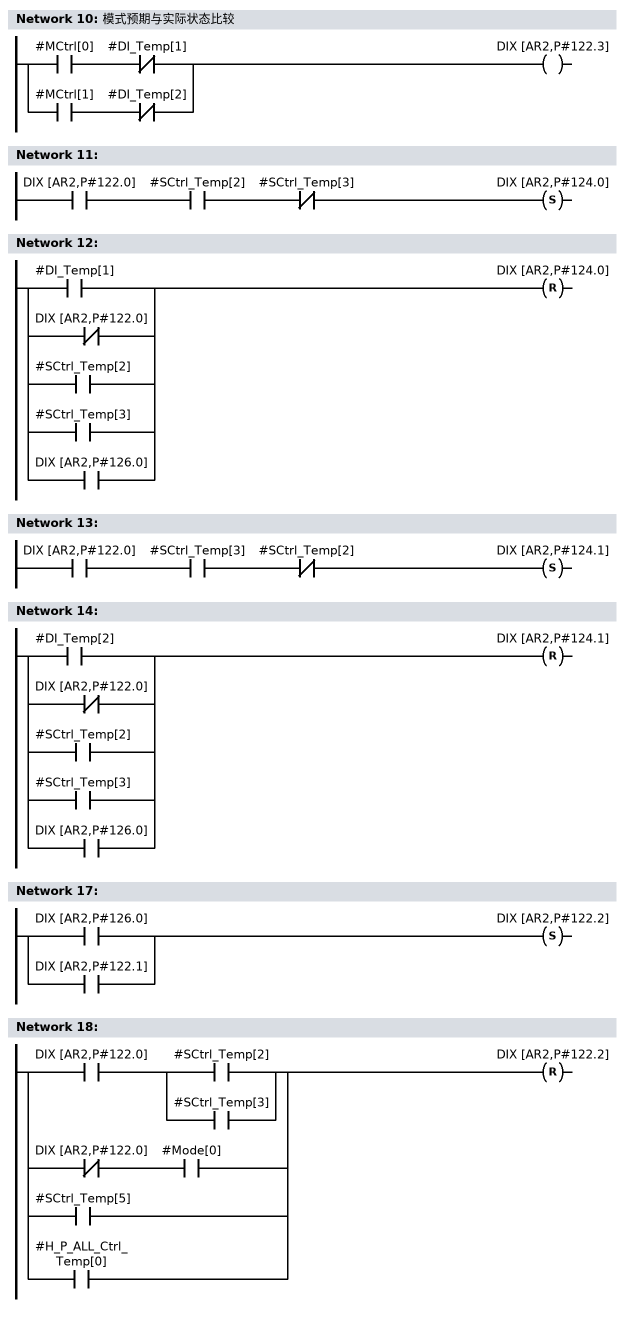
NETWORK
TITLE = 模式预期与实际状态比较
      A     #MCtrl[0];
      AN    #DI_Temp[1];
      O;
      A     #MCtrl[1];
      AN    #DI_Temp[2];
      =     DIX [AR2,P#122.3];
NETWORK
TITLE =
      A     DIX [AR2,P#122.0];
      A     #SCtrl_Temp[2];
      AN    #SCtrl_Temp[3];
      S     DIX [AR2,P#124.0];
NETWORK
TITLE =
      O     #DI_Temp[1];
      ON    DIX [AR2,P#122.0];
      O     #SCtrl_Temp[2];
      O     #SCtrl_Temp[3];
      O     DIX [AR2,P#126.0];
      R     DIX [AR2,P#124.0];
NETWORK
TITLE =
      A     DIX [AR2,P#122.0];
      A     #SCtrl_Temp[3];
      AN    #SCtrl_Temp[2];
      S     DIX [AR2,P#124.1];
NETWORK
TITLE =
      O     #DI_Temp[2];
      ON    DIX [AR2,P#122.0];
      O     #SCtrl_Temp[2];
      O     #SCtrl_Temp[3];
      O     DIX [AR2,P#126.0];
      R     DIX [AR2,P#124.1];
NETWORK
TITLE =
      A(;
      O     DIX [AR2,P#124.0];
      O     DIX [AR2,P#124.1];
      );
      AN    #SCtrl_Temp[2];
      AN    #SCtrl_Temp[3];
      =     L 0.0;
      BLD   103;
      BLD   16;
      =     L 7.0;
      L     DINO;
      T     LW 5;
      CDB;
      OPN   DI [LW 5];
      TAR2  LD 1;
      A     L 0.0;
      =     DIX [AR2,P#34.0];
      L     L#90000;
      T     DID [AR2,P#36.0];
      +AR2  P#34.0;
      UC    "TON";
      LAR2  LD 1;
      A     DIX [AR2,P#40.0];
      =     DBX [AR2,P#126.0];
      CDB;
      BLD   17;
      NOP   0;
NETWORK
TITLE =
      A(;
      O     #DO_Temp[0];
      O     #DO_Temp[1];
      );
      =     L 0.0;
      BLD   103;
      BLD   16;
      =     L 7.0;
      L     DINO;
      T     LW 5;
      CDB;
      OPN   DI [LW 5];
      TAR2  LD 1;
      A     L 0.0;
      =     DIX [AR2,P#56.0];
      L     L#90000;
      T     DID [AR2,P#58.0];
      +AR2  P#56.0;
      UC    "TON";
      LAR2  LD 1;
      A     DIX [AR2,P#62.0];
      =     DBX [AR2,P#122.1];
      CDB;
      BLD   17;
      NOP   0;
NETWORK
TITLE =
      O     DIX [AR2,P#126.0];
      O     DIX [AR2,P#122.1];
      S     DIX [AR2,P#122.2];
NETWORK
TITLE =
      A     DIX [AR2,P#122.0];
      A(;
      O     #SCtrl_Temp[2];
      O     #SCtrl_Temp[3];
      );
      O;
      AN    DIX [AR2,P#122.0];
      A     #Mode[0];
      O     #SCtrl_Temp[5];
      O     #H_P_ALL_Ctrl_Temp[0];
      R     DIX [AR2,P#122.2];
NETWORK
TITLE =
      A(;
      A     #DO_Temp[0];
      A     #DI_Temp[1];
      O;
      A     #DO_Temp[1];
      A     #DI_Temp[2];
      );
      =     L 0.0;
      BLD   103;
      BLD   16;
      =     L 7.0;
      L     DINO;
      T     LW 5;
      CDB;
      OPN   DI [LW 5];
      TAR2  LD 1;
      A     L 0.0;
      =     DIX [AR2,P#78.0];
      L     L#20000;
      T     DID [AR2,P#80.0];
      +AR2  P#78.0;
      UC    "TON";
      LAR2  LD 1;
      A     DIX [AR2,P#84.0];
      =     DBX [AR2,P#29.2];
      CDB;
      BLD   17;
      NOP   0;
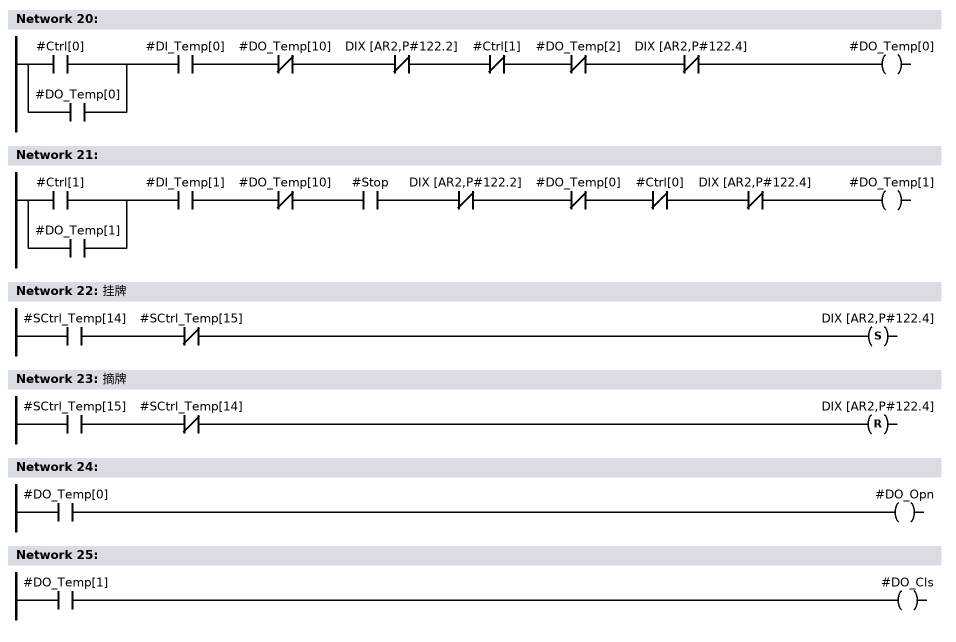
NETWORK
TITLE =
      A(;
      O     #Ctrl[0];
      O     #DO_Temp[0];
      );
      A     #DI_Temp[0];
      AN    #DO_Temp[10];
      AN    DIX [AR2,P#122.2];
      AN    #Ctrl[1];
      AN    #DO_Temp[2];
      AN    DIX [AR2,P#122.4];
      =     #DO_Temp[0];
NETWORK
TITLE =
      A(;
      O     #Ctrl[1];
      O     #DO_Temp[1];
      );
      A     #DI_Temp[1];
      AN    #DO_Temp[10];
      A     #Stop;
      AN    DIX [AR2,P#122.2];
      AN    #DO_Temp[0];
      AN    #Ctrl[0];
      AN    DIX [AR2,P#122.4];
      =     #DO_Temp[1];
NETWORK
TITLE = 挂牌
      A     #SCtrl_Temp[14];
      AN    #SCtrl_Temp[15];
      S     DIX [AR2,P#122.4];
NETWORK
TITLE = 摘牌
      A     #SCtrl_Temp[15];
      AN    #SCtrl_Temp[14];
      R     DIX [AR2,P#122.4];
NETWORK
TITLE =
      A     #DO_Temp[0];
      =     #DO_Opn;
NETWORK
TITLE =
      A     #DO_Temp[1];
      =     #DO_Cls;
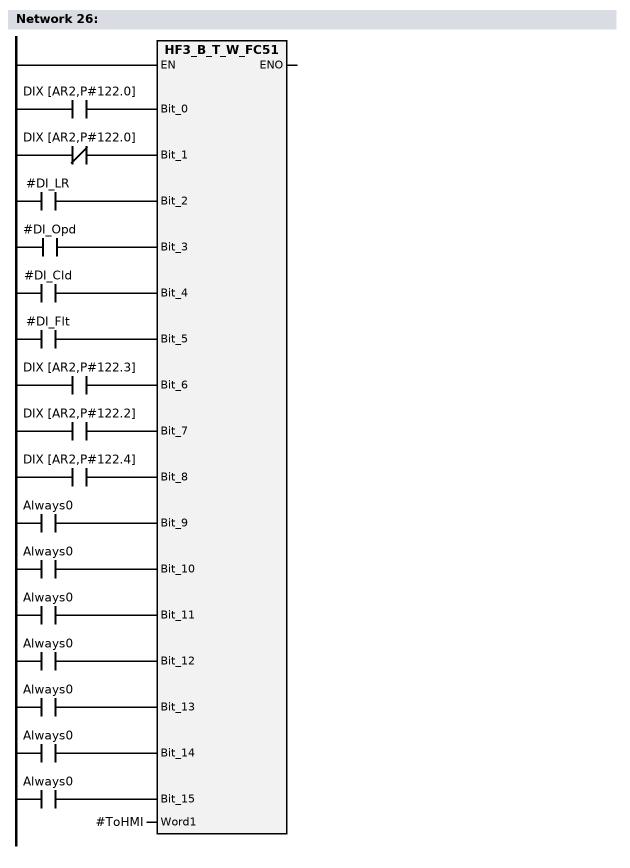
NETWORK
TITLE =
      A     DIX [AR2,P#122.0];
      =     L 0.0;
      BLD   103;
      AN    DIX [AR2,P#122.0];
      =     L 0.1;
      BLD   103;
      A     #DI_LR;
      =     L 0.2;
      BLD   103;
      A     #DI_Opd;
      =     L 0.3;
      BLD   103;
      A     #DI_Cld;
      =     L 0.4;
      BLD   103;
      A     #DI_Flt;
      =     L 0.5;
      BLD   103;
      A     DIX [AR2,P#122.3];
      =     L 0.6;
      BLD   103;
      A     DIX [AR2,P#122.2];
      =     L 0.7;
      BLD   103;
      A     DIX [AR2,P#122.4];
      =     L 1.0;
      BLD   103;
      A     "Always0";
      =     L 1.1;
      BLD   103;
      A     "Always0";
      =     L 1.2;
      BLD   103;
      A     "Always0";
      =     L 1.3;
      BLD   103;
      A     "Always0";
      =     L 1.4;
      BLD   103;
      A     "Always0";
      =     L 1.5;
      BLD   103;
      A     "Always0";
      =     L 1.6;
      BLD   103;
      A     "Always0";
      =     L 1.7;
      BLD   103;
      CALL  "HF3_B_T_W_FC51" (
           Bit_0                    := L 0.0,
           Bit_1                    := L 0.1,
           Bit_2                    := L 0.2,
           Bit_3                    := L 0.3,
           Bit_4                    := L 0.4,
           Bit_5                    := L 0.5,
           Bit_6                    := L 0.6,
           Bit_7                    := L 0.7,
           Bit_8                    := L 1.0,
           Bit_9                    := L 1.1,
           Bit_10                   := L 1.2,
           Bit_11                   := L 1.3,
           Bit_12                   := L 1.4,
           Bit_13                   := L 1.5,
           Bit_14                   := L 1.6,
           Bit_15                   := L 1.7,
           Word1                    := #ToHMI);
      NOP   0;
END_FUNCTION_BLOCK

FUNCTION_BLOCK "HF3_FHF_RFM_FB2811"	// FB 2811
VERSION : 0.1
BEGIN
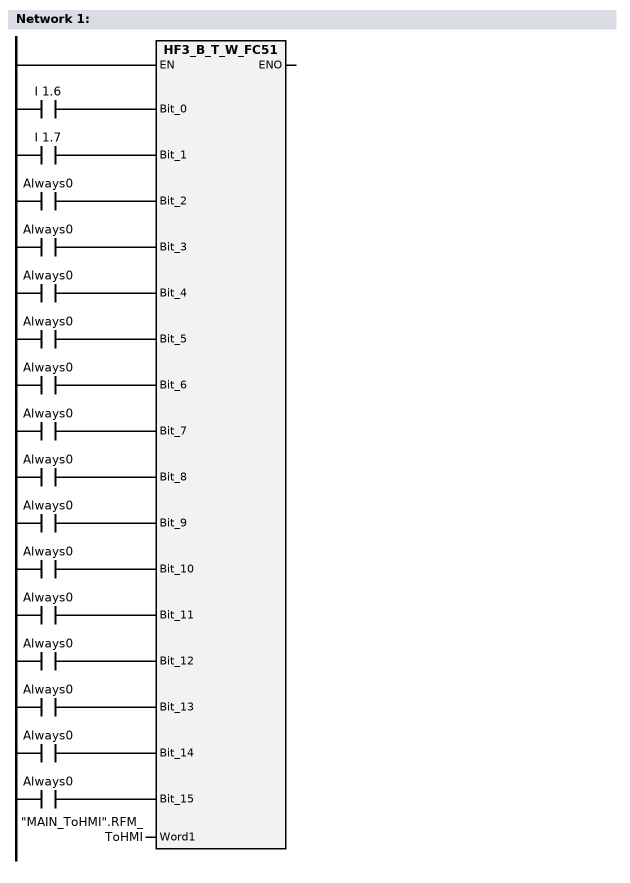
NETWORK
TITLE =
      A     I 1.6;
      =     L 0.0;
      BLD   103;
      A     I 1.7;
      =     L 0.1;
      BLD   103;
      A     "Always0";
      =     L 0.2;
      BLD   103;
      A     "Always0";
      =     L 0.3;
      BLD   103;
      A     "Always0";
      =     L 0.4;
      BLD   103;
      A     "Always0";
      =     L 0.5;
      BLD   103;
      A     "Always0";
      =     L 0.6;
      BLD   103;
      A     "Always0";
      =     L 0.7;
      BLD   103;
      A     "Always0";
      =     L 1.0;
      BLD   103;
      A     "Always0";
      =     L 1.1;
      BLD   103;
      A     "Always0";
      =     L 1.2;
      BLD   103;
      A     "Always0";
      =     L 1.3;
      BLD   103;
      A     "Always0";
      =     L 1.4;
      BLD   103;
      A     "Always0";
      =     L 1.5;
      BLD   103;
      A     "Always0";
      =     L 1.6;
      BLD   103;
      A     "Always0";
      =     L 1.7;
      BLD   103;
      CALL  "HF3_B_T_W_FC51" (
           Bit_0                    := L 0.0,
           Bit_1                    := L 0.1,
           Bit_2                    := L 0.2,
           Bit_3                    := L 0.3,
           Bit_4                    := L 0.4,
           Bit_5                    := L 0.5,
           Bit_6                    := L 0.6,
           Bit_7                    := L 0.7,
           Bit_8                    := L 1.0,
           Bit_9                    := L 1.1,
           Bit_10                   := L 1.2,
           Bit_11                   := L 1.3,
           Bit_12                   := L 1.4,
           Bit_13                   := L 1.5,
           Bit_14                   := L 1.6,
           Bit_15                   := L 1.7,
           Word1                    := "MAIN_ToHMI".RFM_ToHMI);
      NOP   0;
END_FUNCTION_BLOCK

FUNCTION_BLOCK "HF3_Senor_FB2821"	// FB 2821
VERSION : 0.1
VAR
  K4_T_A1 : FB 2822;
  H_A4 : FB 2822;
  H_A5 : FB 2822;
  C_A2 : FB 2822;
  C_A3 : FB 2822;
  C_A4 : FB 2822;
  H_A2 : FB 2822;
  H_A3 : FB 2822;
  K4_H_A1 : FB 2822;
  H_A1 : FB 2822;
  H_A6 : FB 2822;
  H_A7 : FB 2822;
  T_A2 : FB 2822;
END_VAR
BEGIN
NETWORK
TITLE = H-A4
      BLD   14;
      =     L 6.0;
      L     DINO;
      T     LW 4;
      CDB;
      OPN   DI [LW 4];
      TAR2  LD 0;
      L     "H_A4_aiTemp";
      T     DIW [AR2,P#92.0];
      L     "H_A4_aiHumi";
      T     DIW [AR2,P#94.0];
      L     0;
      T     DIW [AR2,P#98.0];
      +AR2  P#92.0;
      UC    "HF3_Sensor_FB2822";
      LAR2  LD 0;
      L     DID [AR2,P#100.0];
      OPN   DI 6004;
      T     DID 194;
      OPN   DI [LW 4];
      L     DID [AR2,P#104.0];
      OPN   DI 6004;
      T     DID 190;
      OPN   DI [LW 4];
      CDB;
      BLD   15;
      NOP   0;
NETWORK
TITLE = H-A5
      BLD   14;
      =     L 6.0;
      L     DINO;
      T     LW 4;
      CDB;
      OPN   DI [LW 4];
      TAR2  LD 0;
      L     "H_A5_aiTemp";
      T     DIW [AR2,P#184.0];
      L     "H_A5_aiHumi";
      T     DIW [AR2,P#186.0];
      L     0;
      T     DIW [AR2,P#190.0];
      +AR2  P#184.0;
      UC    "HF3_Sensor_FB2822";
      LAR2  LD 0;
      L     DID [AR2,P#192.0];
      OPN   DI 6004;
      T     DID 202;
      OPN   DI [LW 4];
      L     DID [AR2,P#196.0];
      OPN   DI 6004;
      T     DID 198;
      OPN   DI [LW 4];
      CDB;
      BLD   15;
      NOP   0;
NETWORK
TITLE = C-A3
      BLD   14;
      =     L 6.0;
      L     DINO;
      T     LW 4;
      CDB;
      OPN   DI [LW 4];
      TAR2  LD 0;
      L     "C_A3_aiCO2";
      T     DIW [AR2,P#372.0];
      L     1;
      T     DIW [AR2,P#374.0];
      +AR2  P#368.0;
      UC    "HF3_Sensor_FB2822";
      LAR2  LD 0;
      L     DID [AR2,P#384.0];
      OPN   DI 6004;
      T     DID 138;
      OPN   DI [LW 4];
      CDB;
      BLD   15;
      NOP   0;
NETWORK
TITLE = K4-T-A1
      BLD   14;
      =     L 6.0;
      L     DINO;
      T     LW 4;
      CDB;
      OPN   DI [LW 4];
      TAR2  LD 0;
      L     "K4_T_A1_aiTemp";
      T     #K4_T_A1.aiTEMP;
      L     "K4_T_A1_aiHumi";
      T     #K4_T_A1.aiHUMI;
      L     0;
      T     #K4_T_A1.CGQ_TYPE;
      +AR2  P#0.0;
      UC    "HF3_Sensor_FB2822";
      LAR2  LD 0;
      L     #K4_T_A1.TEMP;
      OPN   DI 6004;
      T     DID 186;
      OPN   DI [LW 4];
      L     #K4_T_A1.HUMI;
      OPN   DI 6004;
      T     DID 182;
      OPN   DI [LW 4];
      CDB;
      BLD   15;
      NOP   0;
NETWORK
TITLE = H-A2
      BLD   14;
      =     L 6.0;
      L     DINO;
      T     LW 4;
      CDB;
      OPN   DI [LW 4];
      TAR2  LD 0;
      L     "H_A2_aiTemp";
      T     DIW [AR2,P#552.0];
      L     "H_A2_aiHumi";
      T     DIW [AR2,P#554.0];
      L     0;
      T     DIW [AR2,P#558.0];
      +AR2  P#552.0;
      UC    "HF3_Sensor_FB2822";
      LAR2  LD 0;
      L     DID [AR2,P#560.0];
      OPN   DI 6004;
      T     DID 178;
      OPN   DI [LW 4];
      L     DID [AR2,P#564.0];
      OPN   DI 6004;
      T     DID 174;
      OPN   DI [LW 4];
      CDB;
      BLD   15;
      NOP   0;
NETWORK
TITLE = H-A3
      BLD   14;
      =     L 6.0;
      L     DINO;
      T     LW 4;
      CDB;
      OPN   DI [LW 4];
      TAR2  LD 0;
      L     "H_A3_aiTemp";
      T     DIW [AR2,P#644.0];
      L     "H_A3_aiHumi";
      T     DIW [AR2,P#646.0];
      L     0;
      T     DIW [AR2,P#650.0];
      +AR2  P#644.0;
      UC    "HF3_Sensor_FB2822";
      LAR2  LD 0;
      L     DID [AR2,P#652.0];
      OPN   DI 6004;
      T     DID 170;
      OPN   DI [LW 4];
      L     DID [AR2,P#656.0];
      OPN   DI 6004;
      T     DID 166;
      OPN   DI [LW 4];
      CDB;
      BLD   15;
      NOP   0;
NETWORK
TITLE = K4-H-A1
      BLD   14;
      =     L 6.0;
      L     DINO;
      T     LW 4;
      CDB;
      OPN   DI [LW 4];
      TAR2  LD 0;
      L     "K4_H_A1_aiTemp";
      T     DIW [AR2,P#736.0];
      L     "K4_H_A1_aiHumi";
      T     DIW [AR2,P#738.0];
      L     0;
      T     DIW [AR2,P#742.0];
      +AR2  P#736.0;
      UC    "HF3_Sensor_FB2822";
      LAR2  LD 0;
      L     DID [AR2,P#744.0];
      OPN   DI 6004;
      T     DID 162;
      OPN   DI [LW 4];
      L     DID [AR2,P#748.0];
      OPN   DI 6004;
      T     DID 158;
      OPN   DI [LW 4];
      CDB;
      BLD   15;
      NOP   0;
NETWORK
TITLE = H-A1
      BLD   14;
      =     L 6.0;
      L     DINO;
      T     LW 4;
      CDB;
      OPN   DI [LW 4];
      TAR2  LD 0;
      L     "H_A1_aiTemp";
      T     DIW [AR2,P#828.0];
      L     "H_A1_aiHumi";
      T     DIW [AR2,P#830.0];
      L     0;
      T     DIW [AR2,P#834.0];
      +AR2  P#828.0;
      UC    "HF3_Sensor_FB2822";
      LAR2  LD 0;
      L     DID [AR2,P#836.0];
      OPN   DI 6004;
      T     DID 154;
      OPN   DI [LW 4];
      L     DID [AR2,P#840.0];
      OPN   DI 6004;
      T     DID 150;
      OPN   DI [LW 4];
      CDB;
      BLD   15;
      NOP   0;
NETWORK
TITLE = H-A6
      BLD   14;
      =     L 6.0;
      L     DINO;
      T     LW 4;
      CDB;
      OPN   DI [LW 4];
      TAR2  LD 0;
      L     "H_A6_aiTemp";
      T     DIW [AR2,P#920.0];
      L     "H_A6_aiHumi";
      T     DIW [AR2,P#922.0];
      L     0;
      T     DIW [AR2,P#926.0];
      +AR2  P#920.0;
      UC    "HF3_Sensor_FB2822";
      LAR2  LD 0;
      L     DID [AR2,P#928.0];
      OPN   DI 6004;
      T     DID 218;
      OPN   DI [LW 4];
      L     DID [AR2,P#932.0];
      OPN   DI 6004;
      T     DID 214;
      OPN   DI [LW 4];
      CDB;
      BLD   15;
      NOP   0;
NETWORK
TITLE = H-A7
      BLD   14;
      =     L 6.0;
      L     DINO;
      T     LW 4;
      CDB;
      OPN   DI [LW 4];
      TAR2  LD 0;
      L     "H_A7_aiTemp";
      T     DIW [AR2,P#1012.0];
      L     "H_A7_aiHumi";
      T     DIW [AR2,P#1014.0];
      L     0;
      T     DIW [AR2,P#1018.0];
      +AR2  P#1012.0;
      UC    "HF3_Sensor_FB2822";
      LAR2  LD 0;
      L     DID [AR2,P#1020.0];
      OPN   DI 6004;
      T     DID 210;
      OPN   DI [LW 4];
      L     DID [AR2,P#1024.0];
      OPN   DI 6004;
      T     DID 206;
      OPN   DI [LW 4];
      CDB;
      BLD   15;
      NOP   0;
NETWORK
TITLE = C-A2
      BLD   14;
      =     L 6.0;
      L     DINO;
      T     LW 4;
      CDB;
      OPN   DI [LW 4];
      TAR2  LD 0;
      L     "C_A2_aiCO2";
      T     DIW [AR2,P#280.0];
      L     1;
      T     DIW [AR2,P#282.0];
      +AR2  P#276.0;
      UC    "HF3_Sensor_FB2822";
      LAR2  LD 0;
      L     DID [AR2,P#292.0];
      OPN   DI 6004;
      T     DID 134;
      OPN   DI [LW 4];
      CDB;
      BLD   15;
      NOP   0;
NETWORK
TITLE = C-A4
      BLD   14;
      =     L 6.0;
      L     DINO;
      T     LW 4;
      CDB;
      OPN   DI [LW 4];
      TAR2  LD 0;
      L     "C_A4_aiCO2";
      T     DIW [AR2,P#464.0];
      L     1;
      T     DIW [AR2,P#466.0];
      +AR2  P#460.0;
      UC    "HF3_Sensor_FB2822";
      LAR2  LD 0;
      L     DID [AR2,P#476.0];
      OPN   DI 6004;
      T     DID 142;
      OPN   DI [LW 4];
      CDB;
      BLD   15;
      NOP   0;
NETWORK
TITLE = T_A2
      BLD   14;
      =     L 6.0;
      L     DINO;
      T     LW 4;
      CDB;
      OPN   DI [LW 4];
      TAR2  LD 0;
      L     "T_A2_aiTemp";
      T     DIW [AR2,P#1104.0];
      L     "T_A2_aiHumi";
      T     DIW [AR2,P#1106.0];
      L     0;
      T     DIW [AR2,P#1110.0];
      +AR2  P#1104.0;
      UC    "HF3_Sensor_FB2822";
      LAR2  LD 0;
      L     DID [AR2,P#1112.0];
      OPN   DI 6004;
      T     DID 226;
      OPN   DI [LW 4];
      L     DID [AR2,P#1116.0];
      OPN   DI 6004;
      T     DID 222;
      OPN   DI [LW 4];
      CDB;
      BLD   15;
      NOP   0;
END_FUNCTION_BLOCK

FUNCTION_BLOCK "HF3_Sensor_FB2822"	// FB 2822
//know_how_protect
//
AUTHOR : gao
VERSION : 0.1
VAR_INPUT
  aiTEMP : INT ;	//温度反馈
  aiHUMI : INT ;	//湿度反馈
  aiCO2 : INT ;	//二氧化碳反馈
  CGQ_TYPE : INT ;	//所用传感器类型(0)温湿度（1）二氧化碳
END_VAR
VAR_OUTPUT
  TEMP : REAL ;	//温度值
  HUMI : REAL ;	//湿度值
  CO2 : REAL ;	//二氧化碳值
  state_1 : BOOL ;	//线路问题
  state_2 : BOOL ;	//正常
  state_3 : BOOL ;	//读数不正常
END_VAR
VAR
  s2_1 : INT ;	//温湿度
  s2_2 : INT  := 1;	//二氧化碳
  ton1 : SFB 4;
  ton2 : SFB 4;
  ton3 : SFB 4;
END_VAR
VAR_TEMP
  T_BACK_WORD : WORD ;
  T_BWORD_TEMP : INT ;
  end : BOOL ;
  q1 : BOOL ;	//有无信号中间变量
  TH : BOOL ;
  C : BOOL ;
  q2 : BOOL ;	//有无信号中间变量
  q3 : BOOL ;	//有无信号中间变量
  H_BACK_WORD : WORD ;
  C_BACK_WORD : WORD ;
  H_BWORD_TEMP : INT ;
  C_BWORD_TEMP : INT ;
END_VAR
BEGIN
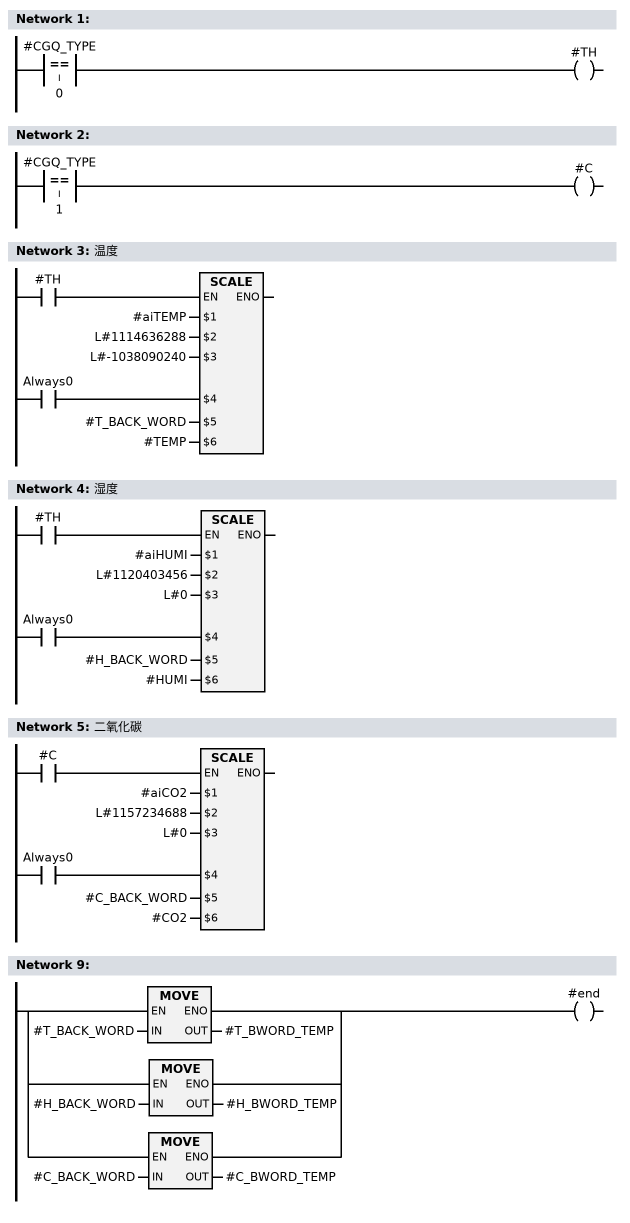
NETWORK
TITLE =
      L     #CGQ_TYPE;
      L     0;
      ==I;
      =     #TH;
NETWORK
TITLE =
      L     #CGQ_TYPE;
      L     1;
      ==I;
      =     #C;
NETWORK
TITLE = 温度
      A     "Always0";
      =     L 14.0;
      BLD   103;
      A     #TH;
      JNB   _001;
      CALL  "SCALE" (
           $1                       := #aiTEMP,
           $2                       := L#1114636288,
           $3                       := L#-1038090240,
           $4                       := L 14.0,
           $5                       := #T_BACK_WORD,
           $6                       := #TEMP);
_001: NOP   0;
NETWORK
TITLE = 湿度
      A     "Always0";
      =     L 14.0;
      BLD   103;
      A     #TH;
      JNB   _002;
      CALL  "SCALE" (
           $1                       := #aiHUMI,
           $2                       := L#1120403456,
           $3                       := L#0,
           $4                       := L 14.0,
           $5                       := #H_BACK_WORD,
           $6                       := #HUMI);
_002: NOP   0;
NETWORK
TITLE = 二氧化碳
      A     "Always0";
      =     L 14.0;
      BLD   103;
      A     #C;
      JNB   _003;
      CALL  "SCALE" (
           $1                       := #aiCO2,
           $2                       := L#1157234688,
           $3                       := L#0,
           $4                       := L 14.0,
           $5                       := #C_BACK_WORD,
           $6                       := #CO2);
_003: NOP   0;
NETWORK
TITLE = 是否接线/模块是否正常（有无信号传输）
      A     #TH;
      A(;
      L     #aiTEMP;
      L     -32768;
      ==I;
      );
      =     L 14.0;
      BLD   103;
      BLD   16;
      =     L 21.0;
      L     DINO;
      T     LW 19;
      CDB;
      OPN   DI [LW 19];
      TAR2  LD 15;
      A     L 14.0;
      =     DIX [AR2,P#26.0];
      L     L#10000;
      T     DID [AR2,P#28.0];
      +AR2  P#26.0;
      UC    "TON";
      LAR2  LD 15;
      A     DIX [AR2,P#32.0];
      =     #q1;
      CDB;
      BLD   17;
      NOP   0;
NETWORK
TITLE =
      A     #TH;
      A(;
      L     #aiHUMI;
      L     -32768;
      ==I;
      );
      =     L 14.0;
      BLD   103;
      BLD   16;
      =     L 21.0;
      L     DINO;
      T     LW 19;
      CDB;
      OPN   DI [LW 19];
      TAR2  LD 15;
      A     L 14.0;
      =     DIX [AR2,P#48.0];
      L     L#10000;
      T     DID [AR2,P#50.0];
      +AR2  P#48.0;
      UC    "TON";
      LAR2  LD 15;
      A     DIX [AR2,P#54.0];
      =     #q2;
      CDB;
      BLD   17;
      NOP   0;
NETWORK
TITLE = 是否接线/模块是否正常（有无信号传输）
      A     #C;
      A(;
      L     #aiCO2;
      L     -32768;
      ==I;
      );
      =     L 14.0;
      BLD   103;
      BLD   16;
      =     L 21.0;
      L     DINO;
      T     LW 19;
      CDB;
      OPN   DI [LW 19];
      TAR2  LD 15;
      A     L 14.0;
      =     DIX [AR2,P#70.0];
      L     L#10000;
      T     DID [AR2,P#72.0];
      +AR2  P#70.0;
      UC    "TON";
      LAR2  LD 15;
      A     DIX [AR2,P#76.0];
      =     #q3;
      CDB;
      BLD   17;
      NOP   0;
NETWORK
TITLE =
      O(;
      L     #T_BACK_WORD;
      T     #T_BWORD_TEMP;
      SET;
      SAVE;
      CLR;
      A     BR;
      );
      O(;
      L     #H_BACK_WORD;
      T     #H_BWORD_TEMP;
      SET;
      SAVE;
      CLR;
      A     BR;
      );
      O(;
      L     #C_BACK_WORD;
      T     #C_BWORD_TEMP;
      SET;
      SAVE;
      CLR;
      A     BR;
      );
      =     #end;
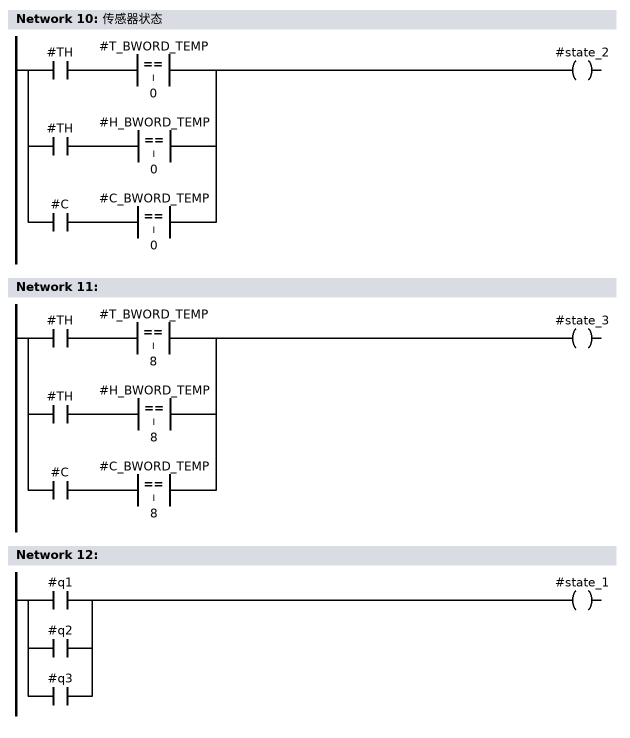
NETWORK
TITLE = 传感器状态
      A     #TH;
      A(;
      L     #T_BWORD_TEMP;
      L     0;
      ==I;
      );
      O;
      A     #TH;
      A(;
      L     #H_BWORD_TEMP;
      L     0;
      ==I;
      );
      O;
      A     #C;
      A(;
      L     #C_BWORD_TEMP;
      L     0;
      ==I;
      );
      =     #state_2;
NETWORK
TITLE =
      A     #TH;
      A(;
      L     #T_BWORD_TEMP;
      L     8;
      ==I;
      );
      O;
      A     #TH;
      A(;
      L     #H_BWORD_TEMP;
      L     8;
      ==I;
      );
      O;
      A     #C;
      A(;
      L     #C_BWORD_TEMP;
      L     8;
      ==I;
      );
      =     #state_3;
NETWORK
TITLE =
      O     #q1;
      O     #q2;
      O     #q3;
      =     #state_1;
END_FUNCTION_BLOCK

FUNCTION_BLOCK "从端与主端通讯"	// FB 2832
VERSION : 0.1
VAR
  A1_B1_CommOK : BOOL ;
  A2_B2_CommOK : BOOL ;
  A_B_Comm : FB 202;
END_VAR
BEGIN
NETWORK
TITLE = B-AͨѶ
      BLD   14;
      =     L 6.0;
      L     DINO;
      T     LW 4;
      CDB;
      OPN   DI [LW 4];
      TAR2  LD 0;
      +AR2  P#2.0;
      UC    "S7400H-COM-SLAVE-MAIN";
      LAR2  LD 0;
      A     #A_B_Comm.STATUS_1;
      =     DBX [AR2,P#0.0];
      A     #A_B_Comm.STATUS_2;
      =     DBX [AR2,P#0.1];
      CDB;
      BLD   15;
      NOP   0;
END_FUNCTION_BLOCK

FUNCTION_BLOCK "HF3_MODE_PRO"	// FB 3000
//模式拆解~ 根据车站实际设备配置
VERSION : 0.1
VAR
  Mode_Explode : FB 3020;
  FC3011_Return : INT ;
  SYS_INT : FB 3007;
END_VAR
BEGIN
NETWORK
TITLE = A端系统模式拆解
// (network holds code this reader does not know; not shown)
NETWORK
TITLE =
      A     "Always0";
      JNB   _001;
      BLD   14;
      =     L 6.0;
      L     DINO;
      T     LW 4;
      CDB;
      OPN   DI [LW 4];
      TAR2  LD 0;
      +AR2  P#364.0;
      UC    FB 3007;
      LAR2  LD 0;
      CDB;
      BLD   15;
_001: NOP   0;
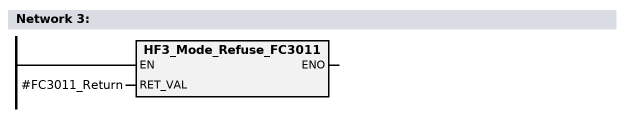
NETWORK
TITLE =
      CALL  "HF3_Mode_Refuse_FC3011" (
           RET_VAL                  := #FC3011_Return);
      NOP   0;
END_FUNCTION_BLOCK

FUNCTION_BLOCK FB 3007
VERSION : 0.0
VAR_OUTPUT
  P_H_Run_Code : ARRAY  [0 .. 40 ] OF INT ;
  P_H_Run_Mod : ARRAY  [0 .. 40 ] OF INT ;
  PT_Mode : ARRAY  [0 .. 40 ] OF TIME ;
  PT01 : TIME ;
  PT02 : TIME ;
  PT03 : TIME ;
  PT04 : TIME ;
  PT05 : TIME ;
  PT06 : TIME ;
  PT07 : TIME ;
  PT08 : TIME ;
  PT09 : TIME ;
  PT10 : TIME ;
  PT11 : TIME ;
  PT12 : TIME ;
  PT13 : TIME ;
  PT14 : TIME ;
  PT15 : TIME ;
  PT16 : TIME ;
  PT17 : TIME ;
  PT18 : TIME ;
  PT19 : TIME ;
  PT20 : TIME ;
  PT21 : TIME ;
  PT22 : TIME ;
  PT23 : TIME ;
  PT24 : TIME ;
  PT25 : TIME ;
  PT26 : TIME ;
  PT27 : TIME ;
  PT28 : TIME ;
END_VAR
VAR
  I : INT ;
  J : INT ;
  N : INT ;
  ton1 : SFB 4;	//Static Variables
  Ton2 : SFB 4;
  ton3 : SFB 4;
  Ton4 : SFB 4;
  ton5 : SFB 4;
  ton6 : SFB 4;
  DevA_SingCtrl : BOOL ;
  DevB_SingCtrl : BOOL ;
  Dev_SingCtrl : BOOL ;	//新增
  H_P_Equ_TSP : ARRAY  [0 .. 40 ] OF TIME ;
  H_P_Mod_TSP : ARRAY  [0 .. 40 ] OF TIME ;
  GrpCtrl_Exist : BOOL ;
END_VAR
BEGIN
// body was compiled from an SCL source; compiled code not shown
END_FUNCTION_BLOCK

FUNCTION_BLOCK "HF3_Mode_Explode_FB3019"	// FB 3020
VERSION : 0.0
VAR_INPUT
  BigA_Act_Mode : STRUCT
   BigA_Mode_Num : INT ;
   WORD0 : WORD ;
   WORD1 : WORD ;
   WORD2 : WORD ;
   WORD3 : WORD ;
   WORD4 : WORD ;
   WORD5 : WORD ;
   WORD6 : WORD ;
   WORD7 : WORD ;
  END_STRUCT ;
  TubA_Act_Mode : STRUCT
   TubA_Mode_Num : INT ;
   WORD0 : WORD ;
   WORD1 : WORD ;
   WORD2 : WORD ;
   WORD3 : WORD ;
   WORD4 : WORD ;
   WORD5 : WORD ;
   WORD6 : WORD ;
   WORD7 : WORD ;
  END_STRUCT ;
  A1_Act_Mode : STRUCT
   A1_Mode_Num : INT ;
   WORD0 : WORD ;
   WORD1 : WORD ;
   WORD2 : WORD ;
   WORD3 : WORD ;
   WORD4 : WORD ;
   WORD5 : WORD ;
   WORD6 : WORD ;
   WORD7 : WORD ;
  END_STRUCT ;
  A2_Act_Mode : STRUCT
   A2_Mode_Num : INT ;
   WORD0 : WORD ;
   WORD1 : WORD ;
   WORD2 : WORD ;
   WORD3 : WORD ;
   WORD4 : WORD ;
   WORD5 : WORD ;
   WORD6 : WORD ;
   WORD7 : WORD ;
  END_STRUCT ;
  A3_Act_Mode : STRUCT
   A3_Mode_Num : INT ;
   WORD0 : WORD ;
   WORD1 : WORD ;
   WORD2 : WORD ;
   WORD3 : WORD ;
   WORD4 : WORD ;
   WORD5 : WORD ;
   WORD6 : WORD ;
   WORD7 : WORD ;
  END_STRUCT ;
  A4_Act_Mode : STRUCT
   A4_Mode_Num : INT ;
   WORD0 : WORD ;
   WORD1 : WORD ;
   WORD2 : WORD ;
   WORD3 : WORD ;
   WORD4 : WORD ;
   WORD5 : WORD ;
   WORD6 : WORD ;
   WORD7 : WORD ;
  END_STRUCT ;
  A5_Act_Mode : STRUCT
   A5_Mode_Num : INT ;
   WORD0 : WORD ;
   WORD1 : WORD ;
   WORD2 : WORD ;
   WORD3 : WORD ;
   WORD4 : WORD ;
   WORD5 : WORD ;
   WORD6 : WORD ;
   WORD7 : WORD ;
  END_STRUCT ;
  A6_Act_Mode : STRUCT
   A6_Mode_Num : INT ;
   WORD0 : WORD ;
   WORD1 : WORD ;
   WORD2 : WORD ;
   WORD3 : WORD ;
   WORD4 : WORD ;
   WORD5 : WORD ;
   WORD6 : WORD ;
   WORD7 : WORD ;
  END_STRUCT ;
  A7_Act_Mode : STRUCT
   A7_Mode_Num : INT ;
   WORD0 : WORD ;
   WORD1 : WORD ;
   WORD2 : WORD ;
   WORD3 : WORD ;
   WORD4 : WORD ;
   WORD5 : WORD ;
   WORD6 : WORD ;
   WORD7 : WORD ;
  END_STRUCT ;
  A8_Act_Mode : STRUCT
   A8_Mode_Num : INT ;
   WORD0 : WORD ;
   WORD1 : WORD ;
   WORD2 : WORD ;
   WORD3 : WORD ;
   WORD4 : WORD ;
   WORD5 : WORD ;
   WORD6 : WORD ;
   WORD7 : WORD ;
  END_STRUCT ;
  A9_Act_Mode : STRUCT
   A9_Mode_Num : INT ;
   WORD0 : WORD ;
   WORD1 : WORD ;
   WORD2 : WORD ;
   WORD3 : WORD ;
   WORD4 : WORD ;
   WORD5 : WORD ;
   WORD6 : WORD ;
   WORD7 : WORD ;
  END_STRUCT ;
  A10_Act_Mode : STRUCT
   A10_Mode_Num : INT ;
   WORD0 : WORD ;
   WORD1 : WORD ;
   WORD2 : WORD ;
   WORD3 : WORD ;
   WORD4 : WORD ;
   WORD5 : WORD ;
   WORD6 : WORD ;
   WORD7 : WORD ;
  END_STRUCT ;
  A11_Act_Mode : STRUCT
   A11_Mode_Num : INT ;
   WORD0 : WORD ;
   WORD1 : WORD ;
   WORD2 : WORD ;
   WORD3 : WORD ;
   WORD4 : WORD ;
   WORD5 : WORD ;
   WORD6 : WORD ;
   WORD7 : WORD ;
  END_STRUCT ;
  A12_Act_Mode : STRUCT
   A12_Mode_Num : INT ;
   WORD0 : WORD ;
   WORD1 : WORD ;
   WORD2 : WORD ;
   WORD3 : WORD ;
   WORD4 : WORD ;
   WORD5 : WORD ;
   WORD6 : WORD ;
   WORD7 : WORD ;
  END_STRUCT ;
END_VAR
VAR_OUTPUT
  KT_A1_Mctrl : ARRAY  [0 .. 3 ] OF BOOL ;
  HPF_A1_Mctrl : ARRAY  [0 .. 3 ] OF BOOL ;
  DTS_A1_Mctrl : ARRAY  [0 .. 3 ] OF BOOL ;
  DTS_A2_Mctrl : ARRAY  [0 .. 3 ] OF BOOL ;
  DTS_A3_Mctrl : ARRAY  [0 .. 3 ] OF BOOL ;
  DTS_A4_Mctrl : ARRAY  [0 .. 3 ] OF BOOL ;
  DTS_A5_Mctrl : ARRAY  [0 .. 3 ] OF BOOL ;
  DTS_A6_Mctrl : ARRAY  [0 .. 3 ] OF BOOL ;
  DPH_A1_Mctrl : ARRAY  [0 .. 3 ] OF BOOL ;
  TVF_A1_Mctrl : ARRAY  [0 .. 3 ] OF BOOL ;
  TVF_A2_Mctrl : ARRAY  [0 .. 3 ] OF BOOL ;
  UOF_A1_Mctrl : ARRAY  [0 .. 3 ] OF BOOL ;
  DM_A1_Mctrl : ARRAY  [0 .. 3 ] OF BOOL ;
  DM_A2_Mctrl : ARRAY  [0 .. 3 ] OF BOOL ;
  DM_A3_Mctrl : ARRAY  [0 .. 3 ] OF BOOL ;
  DM_A4_Mctrl : ARRAY  [0 .. 3 ] OF BOOL ;
  DM_A5_Mctrl : ARRAY  [0 .. 3 ] OF BOOL ;
  DM_A6_Mctrl : ARRAY  [0 .. 3 ] OF BOOL ;
  DM_A7_Mctrl : ARRAY  [0 .. 3 ] OF BOOL ;
  DM_A8_Mctrl : ARRAY  [0 .. 3 ] OF BOOL ;
  UOF_DT_A1_Mctrl : ARRAY  [0 .. 3 ] OF BOOL ;
  UOF_DT_A2_Mctrl : ARRAY  [0 .. 3 ] OF BOOL ;
  UOF_DT_A3_Mctrl : ARRAY  [0 .. 3 ] OF BOOL ;
  UOF_DT_A4_Mctrl : ARRAY  [0 .. 3 ] OF BOOL ;
  K4_XK_A1_Mctrl : ARRAY  [0 .. 3 ] OF BOOL ;
  K4_HPF_A1_Mctrl : ARRAY  [0 .. 3 ] OF BOOL ;
  K4_DTS_A1_Mctrl : ARRAY  [0 .. 3 ] OF BOOL ;
  K4_DTS_A2_Mctrl : ARRAY  [0 .. 3 ] OF BOOL ;
  K4_DTS_A3_Mctrl : ARRAY  [0 .. 3 ] OF BOOL ;
  T6_XSF_A1_Mctrl : ARRAY  [0 .. 3 ] OF BOOL ;
  T6_XPF_A1_Mctrl : ARRAY  [0 .. 3 ] OF BOOL ;
  T6_D_A1_Mctrl : ARRAY  [0 .. 3 ] OF BOOL ;
  T6_D_A2_Mctrl : ARRAY  [0 .. 3 ] OF BOOL ;
  T7_XPF_A1_Mctrl : ARRAY  [0 .. 3 ] OF BOOL ;
  T7_D_A1_Mctrl : ARRAY  [0 .. 3 ] OF BOOL ;
END_VAR
VAR
  BigA_Word0_Temp : ARRAY  [0 .. 15 ] OF BOOL ;
  BigA_Word1_Temp : ARRAY  [0 .. 15 ] OF BOOL ;
  BigA_Word2_Temp : ARRAY  [0 .. 15 ] OF BOOL ;
  BigA_Word3_Temp : ARRAY  [0 .. 15 ] OF BOOL ;
  TubA_Word0_Temp : ARRAY  [0 .. 15 ] OF BOOL ;
  TubA_Word1_Temp : ARRAY  [0 .. 15 ] OF BOOL ;
  TubA_Word2_Temp : ARRAY  [0 .. 15 ] OF BOOL ;
  TubA_Word3_Temp : ARRAY  [0 .. 15 ] OF BOOL ;
  A1_Word0_Temp : ARRAY  [0 .. 15 ] OF BOOL ;
  A1_Word1_Temp : ARRAY  [0 .. 15 ] OF BOOL ;
  A1_Word2_Temp : ARRAY  [0 .. 15 ] OF BOOL ;
  A1_Word3_Temp : ARRAY  [0 .. 15 ] OF BOOL ;
  A2_Word0_Temp : ARRAY  [0 .. 15 ] OF BOOL ;
  A2_Word1_Temp : ARRAY  [0 .. 15 ] OF BOOL ;
  A2_Word2_Temp : ARRAY  [0 .. 15 ] OF BOOL ;
  A2_Word3_Temp : ARRAY  [0 .. 15 ] OF BOOL ;
  A3_Word0_Temp : ARRAY  [0 .. 15 ] OF BOOL ;
  A3_Word1_Temp : ARRAY  [0 .. 15 ] OF BOOL ;
  A3_Word2_Temp : ARRAY  [0 .. 15 ] OF BOOL ;
  A3_Word3_Temp : ARRAY  [0 .. 15 ] OF BOOL ;
END_VAR
BEGIN
// body was compiled from an SCL source; compiled code not shown
END_FUNCTION_BLOCK

FUNCTION "IMCC_Pro" : VOID	// FC 1
VERSION : 0.1
BEGIN
NETWORK
TITLE = cyclic call of FB "MB_PNHCL"- S7 is client
      L     T#1S200MS;
      T     "CONTROL_DAT".RECV_TIMEOUT;
      L     T#5S;
      T     "CONTROL_DAT".CONN_TIMEOUT;
      SET;
      R     "CONTROL_DAT".DISCONNECT;
      CALL  "MB_PNHCL" , "IDB_MODBUS" (
           DIW 0                    := "CONTROL_DAT".id_0_a,
           DIW 2                    := "CONTROL_DAT".id_1_a,
           DIW 8                    := 2,
           DID 10                   := "CONTROL_DAT".reuse_conn_time,
           DIX 14.0                 := "CONTROL_DAT".use_all_conn,
           DID 16                   := "CONTROL_DAT".RECV_TIMEOUT,
           DID 20                   := "CONTROL_DAT".CONN_TIMEOUT,
           DIX 24.0                 := "CONTROL_DAT".DISCONNECT,
           DIW 26                   := 3,
           DIX 28.0                 := "CONTROL_DAT".Init,
           DIX 28.1                 := "CONTROL_DAT".ENQ,
           DIB 29                   := "CONTROL_DAT".DATA_TYPE,
           DIW 30                   := "CONTROL_DAT".START_ADDRESS,
           DIW 32                   := "CONTROL_DAT".LENGTH,
           DIX 34.0                 := "CONTROL_DAT".WRITE_READ,
           DIB 35                   := "CONTROL_DAT".UNIT,
           DIX 36.0                 := "CONTROL_DAT".LICENSED,
           DIX 36.1                 := "CONTROL_DAT".BUSY,
           DIX 36.2                 := "CONTROL_DAT".DONE,
           DIX 36.3                 := "CONTROL_DAT".ERROR,
           DIX 36.4                 := "CONTROL_DAT".ESTAB_0A,
           DIW 38                   := "CONTROL_DAT".STATUS_0A,
           DIX 40.0                 := "CONTROL_DAT".ESTAB_1A,
           DIW 42                   := "CONTROL_DAT".STATUS_1A,
           DIX 72.0                 := "CONTROL_DAT".RedErrS7,
           DIX 72.1                 := "CONTROL_DAT".RedErrDev,
           DIX 72.2                 := "CONTROL_DAT".TotComErr,
           DIX 72.3                 := "CONTROL_DAT".Init_Error,
           DIW 74                   := "CONTROL_DAT".Init_Status);
      A     "CONTROL_DAT".ENQ;
      R     "CONTROL_DAT".ENQ;
      A     "CONTROL_DAT".DONE;
      JCN   err;
      L     "CONTROL_DAT".Count_Done;
      +     1;
      T     "CONTROL_DAT".Count_Done;
      JU    end;
err:  A     "CONTROL_DAT".ERROR;	// reset trigger after job has started
// for cyclic data exchange remove the comment keys
//      A     "CONTROL_DAT".BUSY
//      JC    busy
//      O     "CONTROL_DAT".DONE
//      O     "CONTROL_DAT".ERROR
//      S     "CONTROL_DAT".ENQ
//busy: NOP   0
      JCN   end;
      L     "CONTROL_DAT".Count_Error;
// job finished without error
      +     1;	//for test purposes
      T     "CONTROL_DAT".Count_Error;
      L     "CONTROL_DAT".STATUS_0A;
// you can set the parameters for the next job here
// it is set in comments to give you the possibility to use the variable table 
// for changes during test
//      L     1
//      T     "CONTROL_DAT".UNIT
//      L     3
//      T     "CONTROL_DAT".DATA_TYPE
//      L     800
//      T     "CONTROL_DAT".START_ADDRESS
//      L     5
//      T     "CONTROL_DAT".LENGTH
//      SET   
//      =     "CONTROL_DAT".WRITE_READ
//      SET   
//      =     "CONTROL_DAT".ENQ           // job trigger
      T     "CONTROL_DAT".Save_STATUS_0A;
      L     "CONTROL_DAT".STATUS_1A;
      T     "CONTROL_DAT".Save_STATUS_1A;
// job finished with error
end:  NOP   0;
END_FUNCTION

FUNCTION "HF3_B_T_W_FC51" : VOID	// FC 51
VERSION : 0.0
VAR_INPUT
  Bit_0 : BOOL ;
  Bit_1 : BOOL ;
  Bit_2 : BOOL ;
  Bit_3 : BOOL ;
  Bit_4 : BOOL ;
  Bit_5 : BOOL ;
  Bit_6 : BOOL ;
  Bit_7 : BOOL ;
  Bit_8 : BOOL ;
  Bit_9 : BOOL ;
  Bit_10 : BOOL ;
  Bit_11 : BOOL ;
  Bit_12 : BOOL ;
  Bit_13 : BOOL ;
  Bit_14 : BOOL ;
  Bit_15 : BOOL ;
END_VAR
VAR_OUTPUT
  Word1 : WORD ;
END_VAR
VAR_TEMP
  Word2 : WORD ;
END_VAR
BEGIN
// body was compiled from an SCL source; compiled code not shown
END_FUNCTION

FUNCTION "HF3_W_T_B_FC54" : VOID	// FC 54
VERSION : 0.0
VAR_INPUT
  WORD1 : WORD ;
END_VAR
VAR_OUTPUT
  bool1 : ARRAY  [0 .. 15 ] OF
  BOOL ;
END_VAR
BEGIN
NETWORK
TITLE = SCL network
//compiled by SCL compiler version:  SCLCOMP K05.03.07.00_01.02.00.01 release
      SET;
      SAVE;
      =     L 0.1;
      L     #WORD1;
      L     W#16#1;
      AW;
      L     W#16#0;
      <>I;
      BLD   5;
      T     LD 3;
      TAK;
      T     LD 7;
      L     P##bool1;
      LAR1;
      L     W [AR1,P#0.0];
      T     LW 1;
      OPN   DB [LW 1];
      L     D [AR1,P#2.0];
      LAR1;
      L     LD 7;
      L     LD 3;
      =      [AR1,P#0.0];
      L     #WORD1;
      L     W#16#2;
      AW;
      L     W#16#0;
      <>I;
      BLD   5;
      T     LD 3;
      TAK;
      T     LD 7;
      L     P##bool1;
      LAR1;
      L     W [AR1,P#0.0];
      T     LW 1;
      OPN   DB [LW 1];
      L     D [AR1,P#2.0];
      LAR1;
      L     LD 7;
      L     LD 3;
      =      [AR1,P#0.1];
      L     #WORD1;
      L     W#16#4;
      AW;
      L     W#16#0;
      <>I;
      BLD   5;
      T     LD 3;
      TAK;
      T     LD 7;
      L     P##bool1;
      LAR1;
      L     W [AR1,P#0.0];
      T     LW 1;
      OPN   DB [LW 1];
      L     D [AR1,P#2.0];
      LAR1;
      L     LD 7;
      L     LD 3;
      =      [AR1,P#0.2];
      L     #WORD1;
      L     W#16#8;
      AW;
      L     W#16#0;
      <>I;
      BLD   5;
      T     LD 3;
      TAK;
      T     LD 7;
      L     P##bool1;
      LAR1;
      L     W [AR1,P#0.0];
      T     LW 1;
      OPN   DB [LW 1];
      L     D [AR1,P#2.0];
      LAR1;
      L     LD 7;
      L     LD 3;
      =      [AR1,P#0.3];
      L     #WORD1;
      L     W#16#10;
      AW;
      L     W#16#0;
      <>I;
      BLD   5;
      T     LD 3;
      TAK;
      T     LD 7;
      L     P##bool1;
      LAR1;
      L     W [AR1,P#0.0];
      T     LW 1;
      OPN   DB [LW 1];
      L     D [AR1,P#2.0];
      LAR1;
      L     LD 7;
      L     LD 3;
      =      [AR1,P#0.4];
      L     #WORD1;
      L     W#16#20;
      AW;
      L     W#16#0;
      <>I;
      BLD   5;
      T     LD 3;
      TAK;
      T     LD 7;
      L     P##bool1;
      LAR1;
      L     W [AR1,P#0.0];
      T     LW 1;
      OPN   DB [LW 1];
      L     D [AR1,P#2.0];
      LAR1;
      L     LD 7;
      L     LD 3;
      =      [AR1,P#0.5];
      L     #WORD1;
      L     W#16#40;
      AW;
      L     W#16#0;
      <>I;
      BLD   5;
      T     LD 3;
      TAK;
      T     LD 7;
      L     P##bool1;
      LAR1;
      L     W [AR1,P#0.0];
      T     LW 1;
      OPN   DB [LW 1];
      L     D [AR1,P#2.0];
      LAR1;
      L     LD 7;
      L     LD 3;
      =      [AR1,P#0.6];
      L     #WORD1;
      L     W#16#80;
      AW;
      L     W#16#0;
      <>I;
      BLD   5;
      T     LD 3;
      TAK;
      T     LD 7;
      L     P##bool1;
      LAR1;
      L     W [AR1,P#0.0];
      T     LW 1;
      OPN   DB [LW 1];
      L     D [AR1,P#2.0];
      LAR1;
      L     LD 7;
      L     LD 3;
      =      [AR1,P#0.7];
      L     #WORD1;
      L     W#16#100;
      AW;
      L     W#16#0;
      <>I;
      BLD   5;
      T     LD 3;
      TAK;
      T     LD 7;
      L     P##bool1;
      LAR1;
      L     W [AR1,P#0.0];
      T     LW 1;
      OPN   DB [LW 1];
      L     D [AR1,P#2.0];
      LAR1;
      L     LD 7;
      L     LD 3;
      =      [AR1,P#1.0];
      L     #WORD1;
      L     W#16#200;
      AW;
      L     W#16#0;
      <>I;
      BLD   5;
      T     LD 3;
      TAK;
      T     LD 7;
      L     P##bool1;
      LAR1;
      L     W [AR1,P#0.0];
      T     LW 1;
      OPN   DB [LW 1];
      L     D [AR1,P#2.0];
      LAR1;
      L     LD 7;
      L     LD 3;
      =      [AR1,P#1.1];
      L     #WORD1;
      L     W#16#400;
      AW;
      L     W#16#0;
      <>I;
      BLD   5;
      T     LD 3;
      TAK;
      T     LD 7;
      L     P##bool1;
      LAR1;
      L     W [AR1,P#0.0];
      T     LW 1;
      OPN   DB [LW 1];
      L     D [AR1,P#2.0];
      LAR1;
      L     LD 7;
      L     LD 3;
      =      [AR1,P#1.2];
      L     #WORD1;
      L     W#16#800;
      AW;
      L     W#16#0;
      <>I;
      BLD   5;
      T     LD 3;
      TAK;
      T     LD 7;
      L     P##bool1;
      LAR1;
      L     W [AR1,P#0.0];
      T     LW 1;
      OPN   DB [LW 1];
      L     D [AR1,P#2.0];
      LAR1;
      L     LD 7;
      L     LD 3;
      =      [AR1,P#1.3];
      L     #WORD1;
      L     W#16#1000;
      AW;
      L     W#16#0;
      <>I;
      BLD   5;
      T     LD 3;
      TAK;
      T     LD 7;
      L     P##bool1;
      LAR1;
      L     W [AR1,P#0.0];
      T     LW 1;
      OPN   DB [LW 1];
      L     D [AR1,P#2.0];
      LAR1;
      L     LD 7;
      L     LD 3;
      =      [AR1,P#1.4];
      L     #WORD1;
      L     W#16#2000;
      AW;
      L     W#16#0;
      <>I;
      BLD   5;
      T     LD 3;
      TAK;
      T     LD 7;
      L     P##bool1;
      LAR1;
      L     W [AR1,P#0.0];
      T     LW 1;
      OPN   DB [LW 1];
      L     D [AR1,P#2.0];
      LAR1;
      L     LD 7;
      L     LD 3;
      =      [AR1,P#1.5];
      L     #WORD1;
      L     W#16#4000;
      AW;
      L     W#16#0;
      <>I;
      BLD   5;
      T     LD 3;
      TAK;
      T     LD 7;
      L     P##bool1;
      LAR1;
      L     W [AR1,P#0.0];
      T     LW 1;
      OPN   DB [LW 1];
      L     D [AR1,P#2.0];
      LAR1;
      L     LD 7;
      L     LD 3;
      =      [AR1,P#1.6];
      L     #WORD1;
      L     W#16#8000;
      AW;
      L     W#16#0;
      <>I;
      BLD   5;
      T     LD 3;
      TAK;
      T     LD 7;
      L     P##bool1;
      LAR1;
      L     W [AR1,P#0.0];
      T     LW 1;
      OPN   DB [LW 1];
      L     D [AR1,P#2.0];
      LAR1;
      L     LD 7;
      L     LD 3;
      =      [AR1,P#1.7];
      A     L 0.1;
      SAVE;
      BE;
END_FUNCTION

FUNCTION FC 55 : VOID
VERSION : 0.0
VAR_INPUT
  byte1 : BYTE ;
END_VAR
VAR_OUTPUT
  bit : ARRAY  [0 .. 7 ] OF BOOL ;
END_VAR
BEGIN
// body was compiled from an SCL source; compiled code not shown
END_FUNCTION

FUNCTION FC 59 : VOID
VERSION : 0.0
VAR_INPUT
  IN1 : ARRAY  [0 .. 19 ] OF WORD ;
END_VAR
VAR_OUTPUT
  out1 : INT ;
  out2 : INT ;
  out3 : INT ;
  out4 : INT ;
  out5 : INT ;
  out6 : INT ;
  out7 : INT ;
  out8 : INT ;
  out9 : INT ;
  out10 : INT ;
  out11 : INT ;
  out12 : INT ;
  out13 : INT ;
  out14 : INT ;
  out15 : INT ;
END_VAR
BEGIN
// body was compiled from an SCL source; compiled code not shown
END_FUNCTION

// FC 105: know-how protected block, not included

// FC 106: know-how protected block, not included

FUNCTION "MK_ERROR_SAVE_RACK0" : VOID	// FC 201
VERSION : 0.0
BEGIN
// body was compiled from an SCL source; compiled code not shown
END_FUNCTION

FUNCTION "RIO_Information" : VOID	// FC 202
VERSION : 0.1
BEGIN
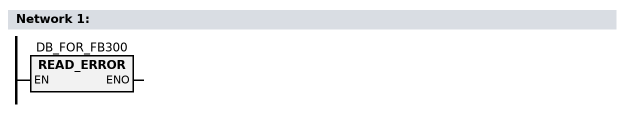
NETWORK
TITLE =
      CALL  "READ_ERROR" , "DB_FOR_FB300";
      NOP   0;
NETWORK
TITLE =
// (network holds code this reader does not know; not shown)
END_FUNCTION

FUNCTION "MK_ERROR_SAVE_RACK1" : VOID	// FC 203
VERSION : 0.0
BEGIN
// body was compiled from an SCL source; compiled code not shown
END_FUNCTION

FUNCTION "DP_ERROR_TO_DB701" : VOID	// FC 204
VERSION : 0.0
VAR_TEMP
  I : INT ;
  J : INT ;
END_VAR
BEGIN
// body was compiled from an SCL source; compiled code not shown
END_FUNCTION

// FC 501: know-how protected block, not included

FUNCTION "BAS_CLOCK" : VOID	// FC 505
TITLE = 校时程序
VERSION : 0.1
VAR_TEMP
  RET1 : INT ;
  RET2 : INT ;
  RET3 : INT ;
END_VAR
BEGIN
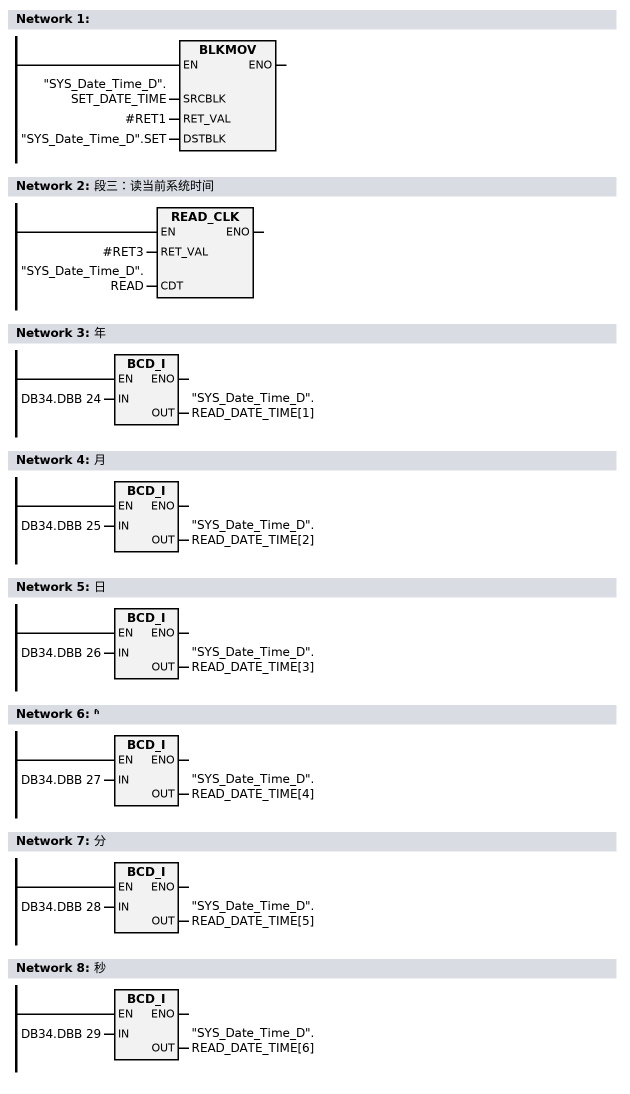
NETWORK
TITLE =
      CALL  "BLKMOV" (
           SRCBLK                   := "SYS_Date_Time_D".SET_DATE_TIME,
           RET_VAL                  := #RET1,
           DSTBLK                   := "SYS_Date_Time_D".SET);
      NOP   0;
NETWORK
TITLE = 段三：读当前系统时间
      CALL  "READ_CLK" (
           RET_VAL                  := #RET3,
           CDT                      := "SYS_Date_Time_D".READ);
      NOP   0;
NETWORK
TITLE = 年
      L     DB34.DBB 24;
      BTI;
      T     "SYS_Date_Time_D".READ_DATE_TIME[1];
NETWORK
TITLE = 月
      L     DB34.DBB 25;
      BTI;
      T     "SYS_Date_Time_D".READ_DATE_TIME[2];
NETWORK
TITLE = 日
      L     DB34.DBB 26;
      BTI;
      T     "SYS_Date_Time_D".READ_DATE_TIME[3];
NETWORK
TITLE = ʱ
      L     DB34.DBB 27;
      BTI;
      T     "SYS_Date_Time_D".READ_DATE_TIME[4];
NETWORK
TITLE = 分
      L     DB34.DBB 28;
      BTI;
      T     "SYS_Date_Time_D".READ_DATE_TIME[5];
NETWORK
TITLE = 秒
      L     DB34.DBB 29;
      BTI;
      T     "SYS_Date_Time_D".READ_DATE_TIME[6];
NETWORK
TITLE =
      L     "SYS_Date_Time_D".READ_DATE_TIME[4];
      L     100;
      *I;
      L     "SYS_Date_Time_D".READ_DATE_TIME[5];
      +I;
      T     "SYS_Date_Time_D".TIME_HM;	/////hour*100+minute
END_FUNCTION

FUNCTION "CPU_Information" : VOID	// FC 523
VERSION : 0.1
VAR_TEMP
  length : STRUCT
   size : WORD ;
   number : WORD ;
  END_STRUCT ;
  length_1 : STRUCT
   size : WORD ;
   number : WORD ;
  END_STRUCT ;
END_VAR
BEGIN
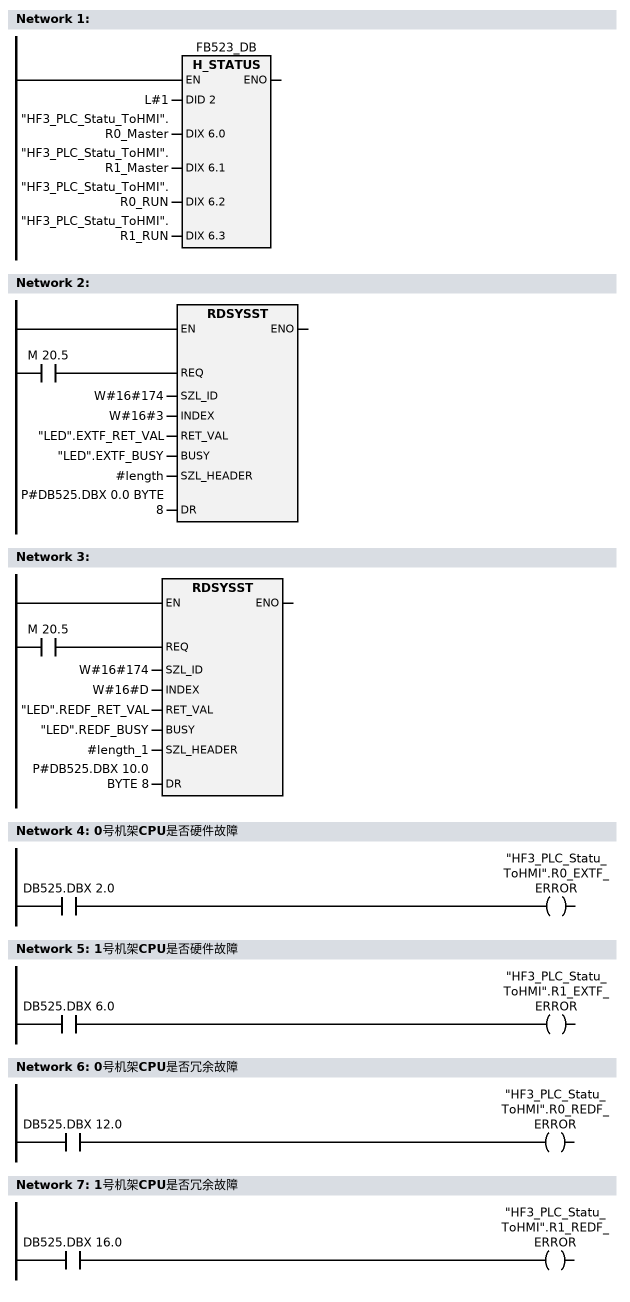
NETWORK
TITLE =
      CALL  "H_STATUS" , "FB523_DB" (
           DID 2                    := L#1,
           DIX 6.0                  := "HF3_PLC_Statu_ToHMI".R0_Master,
           DIX 6.1                  := "HF3_PLC_Statu_ToHMI".R1_Master,
           DIX 6.2                  := "HF3_PLC_Statu_ToHMI".R0_RUN,
           DIX 6.3                  := "HF3_PLC_Statu_ToHMI".R1_RUN);
      NOP   0;
NETWORK
TITLE =
      A     M 20.5;
      =     L 8.0;
      BLD   103;
      CALL  "RDSYSST" (
           REQ                      := L 8.0,
           SZL_ID                   := W#16#174,
           INDEX                    := W#16#3,
           RET_VAL                  := "LED".EXTF_RET_VAL,
           BUSY                     := "LED".EXTF_BUSY,
           SZL_HEADER               := #length,
           DR                       := P#DB525.DBX 0.0 BYTE 8);
      NOP   0;
NETWORK
TITLE =
      A     M 20.5;
      =     L 8.0;
      BLD   103;
      CALL  "RDSYSST" (
           REQ                      := L 8.0,
           SZL_ID                   := W#16#174,
           INDEX                    := W#16#D,
           RET_VAL                  := "LED".REDF_RET_VAL,
           BUSY                     := "LED".REDF_BUSY,
           SZL_HEADER               := #length_1,
           DR                       := P#DB525.DBX 10.0 BYTE 8);
      NOP   0;
NETWORK
TITLE = 0号机架CPU是否硬件故障
      A     DB525.DBX 2.0;
      =     "HF3_PLC_Statu_ToHMI".R0_EXTF_ERROR;
NETWORK
TITLE = 1号机架CPU是否硬件故障
      A     DB525.DBX 6.0;
      =     "HF3_PLC_Statu_ToHMI".R1_EXTF_ERROR;
NETWORK
TITLE = 0号机架CPU是否冗余故障
      A     DB525.DBX 12.0;
      =     "HF3_PLC_Statu_ToHMI".R0_REDF_ERROR;
NETWORK
TITLE = 1号机架CPU是否冗余故障
      A     DB525.DBX 16.0;
      =     "HF3_PLC_Statu_ToHMI".R1_REDF_ERROR;
END_FUNCTION

FUNCTION "ABS_I" : VOID	// FC 1234
VERSION : 0.0
VAR_INPUT
  IN : INT ;
END_VAR
VAR_OUTPUT
  OUT : INT ;
END_VAR
BEGIN
// body was compiled from an SCL source; compiled code not shown
END_FUNCTION

FUNCTION "real_to_int" : VOID	// FC 2000
VERSION : 0.0
VAR_INPUT
  IN : REAL ;
END_VAR
VAR_OUTPUT
  OUT : INT ;
END_VAR
BEGIN
// body was compiled from an SCL source; compiled code not shown
END_FUNCTION

FUNCTION "HF3_IMCC_FC2511" : VOID	// FC 2511
VERSION : 0.1
BEGIN
NETWORK
TITLE = cyclic call of FB "MB_PNHCL"- S7 is client
      L     T#1S200MS;
      T     "CONTROL_DAT".RECV_TIMEOUT;
      L     T#5S;
      T     "CONTROL_DAT".CONN_TIMEOUT;
      SET;
      R     "CONTROL_DAT".DISCONNECT;
      CALL  "MB_PNHCL" , "IDB_MODBUS" (
           DIW 0                    := "CONTROL_DAT".id_0_a,
           DIW 2                    := "CONTROL_DAT".id_1_a,
           DIW 8                    := 2,
           DID 10                   := "CONTROL_DAT".reuse_conn_time,
           DIX 14.0                 := "CONTROL_DAT".use_all_conn,
           DID 16                   := "CONTROL_DAT".RECV_TIMEOUT,
           DID 20                   := "CONTROL_DAT".CONN_TIMEOUT,
           DIX 24.0                 := "CONTROL_DAT".DISCONNECT,
           DIW 26                   := 3,
           DIX 28.0                 := "CONTROL_DAT".Init,
           DIX 28.1                 := "CONTROL_DAT".ENQ,
           DIB 29                   := "CONTROL_DAT".DATA_TYPE,
           DIW 30                   := "CONTROL_DAT".START_ADDRESS,
           DIW 32                   := "CONTROL_DAT".LENGTH,
           DIX 34.0                 := "CONTROL_DAT".WRITE_READ,
           DIB 35                   := "CONTROL_DAT".UNIT,
           DIX 36.0                 := "CONTROL_DAT".LICENSED,
           DIX 36.1                 := "CONTROL_DAT".BUSY,
           DIX 36.2                 := "CONTROL_DAT".DONE,
           DIX 36.3                 := "CONTROL_DAT".ERROR,
           DIX 36.4                 := "CONTROL_DAT".ESTAB_0A,
           DIW 38                   := "CONTROL_DAT".STATUS_0A,
           DIX 40.0                 := "CONTROL_DAT".ESTAB_1A,
           DIW 42                   := "CONTROL_DAT".STATUS_1A,
           DIX 72.0                 := "CONTROL_DAT".RedErrS7,
           DIX 72.1                 := "CONTROL_DAT".RedErrDev,
           DIX 72.2                 := "CONTROL_DAT".TotComErr,
           DIX 72.3                 := "CONTROL_DAT".Init_Error,
           DIW 74                   := "CONTROL_DAT".Init_Status);
      A     "CONTROL_DAT".ENQ;
      R     "CONTROL_DAT".ENQ;
      A     "CONTROL_DAT".DONE;
      JCN   err;
      L     "CONTROL_DAT".Count_Done;
      +     1;
      T     "CONTROL_DAT".Count_Done;
      JU    end;
err:  A     "CONTROL_DAT".ERROR;	// reset trigger after job has started
// for cyclic data exchange remove the comment keys
//      A     "CONTROL_DAT".BUSY
//      JC    busy
//      O     "CONTROL_DAT".DONE
//      O     "CONTROL_DAT".ERROR
//      S     "CONTROL_DAT".ENQ
//busy: NOP   0
      JCN   end;
      L     "CONTROL_DAT".Count_Error;
// job finished without error
      +     1;	//for test purposes
      T     "CONTROL_DAT".Count_Error;
      L     "CONTROL_DAT".STATUS_0A;
// you can set the parameters for the next job here
// it is set in comments to give you the possibility to use the variable table 
// for changes during test
//      L     1
//      T     "CONTROL_DAT".UNIT
//      L     3
//      T     "CONTROL_DAT".DATA_TYPE
//      L     800
//      T     "CONTROL_DAT".START_ADDRESS
//      L     5
//      T     "CONTROL_DAT".LENGTH
//      SET   
//      =     "CONTROL_DAT".WRITE_READ
//      SET   
//      =     "CONTROL_DAT".ENQ           // job trigger
      T     "CONTROL_DAT".Save_STATUS_0A;
      L     "CONTROL_DAT".STATUS_1A;
      T     "CONTROL_DAT".Save_STATUS_1A;
// job finished with error
end:  NOP   0;
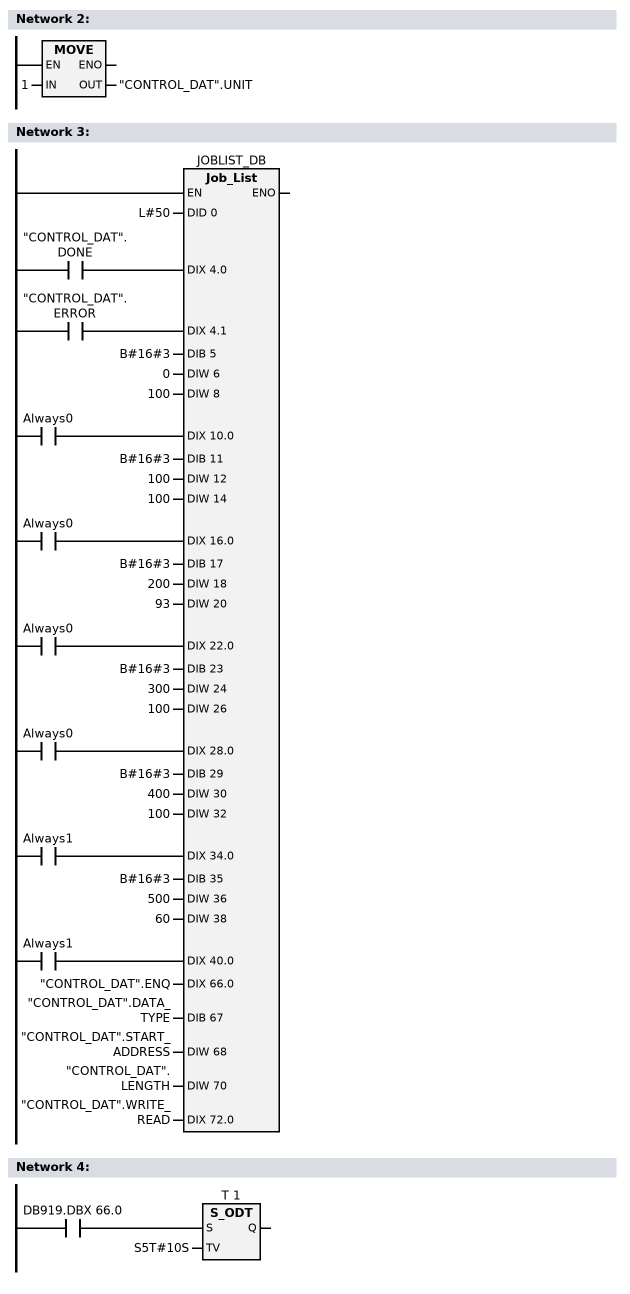
NETWORK
TITLE =
      L     1;
      T     "CONTROL_DAT".UNIT;
      NOP   0;
NETWORK
TITLE =
      A     "CONTROL_DAT".DONE;
      =     L 0.0;
      BLD   103;
      A     "CONTROL_DAT".ERROR;
      =     L 0.1;
      BLD   103;
      A     "Always0";
      =     L 0.2;
      BLD   103;
      A     "Always0";
      =     L 0.3;
      BLD   103;
      A     "Always0";
      =     L 0.4;
      BLD   103;
      A     "Always0";
      =     L 0.5;
      BLD   103;
      A     "Always1";
      =     L 0.6;
      BLD   103;
      A     "Always1";
      =     L 0.7;
      BLD   103;
      CALL  "Job_List" , "JOBLIST_DB" (
           DID 0                    := L#50,
           DIX 4.0                  := L 0.0,
           DIX 4.1                  := L 0.1,
           DIB 5                    := B#16#3,
           DIW 6                    := 0,
           DIW 8                    := 100,
           DIX 10.0                 := L 0.2,
           DIB 11                   := B#16#3,
           DIW 12                   := 100,
           DIW 14                   := 100,
           DIX 16.0                 := L 0.3,
           DIB 17                   := B#16#3,
           DIW 18                   := 200,
           DIW 20                   := 93,
           DIX 22.0                 := L 0.4,
           DIB 23                   := B#16#3,
           DIW 24                   := 300,
           DIW 26                   := 100,
           DIX 28.0                 := L 0.5,
           DIB 29                   := B#16#3,
           DIW 30                   := 400,
           DIW 32                   := 100,
           DIX 34.0                 := L 0.6,
           DIB 35                   := B#16#3,
           DIW 36                   := 500,
           DIW 38                   := 60,
           DIX 40.0                 := L 0.7,
           DIX 66.0                 := "CONTROL_DAT".ENQ,
           DIB 67                   := "CONTROL_DAT".DATA_TYPE,
           DIW 68                   := "CONTROL_DAT".START_ADDRESS,
           DIW 70                   := "CONTROL_DAT".LENGTH,
           DIX 72.0                 := "CONTROL_DAT".WRITE_READ);
      NOP   0;
NETWORK
TITLE =
      A     DB919.DBX 66.0;
      L     S5T#10S;
      SD    T 1;
      NOP   0;
      NOP   0;
      NOP   0;
      NOP   0;
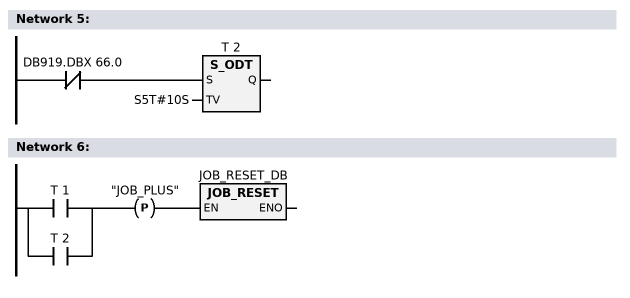
NETWORK
TITLE =
      AN    DB919.DBX 66.0;
      L     S5T#10S;
      SD    T 2;
      NOP   0;
      NOP   0;
      NOP   0;
      NOP   0;
NETWORK
TITLE =
      A(;
      O     T 1;
      O     T 2;
      );
      FP    "JOB_PLUS";
      JNB   _001;
      CALL  "JOB_RESET" , "JOB_RESET_DB";
_001: NOP   0;
END_FUNCTION

FUNCTION "HF3_Mode_Refuse_FC3011" : INT	// FC 3011
VERSION : 0.0
VAR_OUTPUT
  RET_VAL : INT ;
END_VAR
BEGIN
// body was compiled from an SCL source; compiled code not shown
END_FUNCTION

FUNCTION "FUZHI" : VOID	// FC 4000
VERSION : 0.0
BEGIN
// body was compiled from an SCL source; compiled code not shown
END_FUNCTION

